LIN {X 0,Y 740.336,Z 905.286,A -85,B 0,C 180,E1 33713.646,E2 33713.646} C_VEL
LIN {X 0,Y 741.074,Z 665.697,A -85,B 0,C 180,E1 33710.789,E2 33710.789} C_VEL
LIN {X 0,Y 741.733,Z 456.435,A -85,B 0,C 180,E1 33708.221,E2 33708.221} C_VEL
LIN {X 0,Y 741.657,Z 433.468,A -85,B 0,C 180,E1 33707.923,E2 33707.923} C_VEL
LIN {X 0,Y 740.112,Z 427.36,A -85,B 0,C 180,E1 33707.725,E2 33707.725} C_VEL
LIN {X 0,Y 740.318,Z 399.493,A -85,B 0,C 180,E1 33705.878,E2 33705.878} C_VEL
LIN {X 0,Y 737.201,Z 392.802,A -85,B 0,C 180,E1 33705.183,E2 33705.183} C_VEL
LIN {X 0,Y 736.058,Z 389.544,A -85,B 0,C 180,E1 33704.846,E2 33704.846} C_VEL
LIN {X 0,Y 736.094,Z 389.54,A -85,B 0,C 180,E1 33701.833,E2 33701.833} C_VEL
LIN {X 0,Y 736.034,Z 389.542,A -85,B 0,C 180,E1 33699.075,E2 33699.075} C_VEL
LIN {X 0,Y 736.07,Z 389.535,A -85,B 0,C 180,E1 33696.415,E2 33696.415} C_VEL
LIN {X 0,Y 736.045,Z 389.543,A -85,B 0,C 180,E1 33693.349,E2 33693.349} C_VEL
LIN {X 0,Y 736.022,Z 389.539,A -85,B 0,C 180,E1 33690.808,E2 33690.808} C_VEL
LIN {X 0,Y 736.056,Z 389.537,A -85,B 0,C 180,E1 33688.212,E2 33688.212} C_VEL
LIN {X 0,Y 736.036,Z 389.54,A -85,B 0,C 180,E1 33685.164,E2 33685.164} C_VEL
LIN {X 0,Y 736.009,Z 389.543,A -85,B 0,C 180,E1 33682.695,E2 33682.695} C_VEL
LIN {X 0,Y 736.01,Z 389.536,A -85,B 0,C 180,E1 33680.352,E2 33680.352} C_VEL
LIN {X 0,Y 736.099,Z 389.541,A -85,B 0,C 180,E1 33677.55,E2 33677.55} C_VEL
LIN {X 0,Y 736.004,Z 389.539,A -85,B 0,C 180,E1 33674.717,E2 33674.717} C_VEL
LIN {X 0,Y 735.992,Z 389.544,A -85,B 0,C 180,E1 33672.475,E2 33672.475} C_VEL
LIN {X 0,Y 735.989,Z 389.542,A -85,B 0,C 180,E1 33670.173,E2 33670.173} C_VEL
LIN {X 0,Y 736.026,Z 389.541,A -85,B 0,C 180,E1 33667.651,E2 33667.651} C_VEL
LIN {X 0,Y 736.016,Z 389.541,A -85,B 0,C 180,E1 33664.675,E2 33664.675} C_VEL
LIN {X 0,Y 735.992,Z 389.54,A -85,B 0,C 180,E1 33662.258,E2 33662.258} C_VEL
LIN {X 0,Y 735.996,Z 389.544,A -85,B 0,C 180,E1 33660,E2 33660} C_VEL
LIN {X 0,Y 736.012,Z 389.54,A -85,B 0,C 180,E1 33657.664,E2 33657.664} C_VEL
LIN {X 0,Y 736.088,Z 389.541,A -85,B 0,C 180,E1 33654.778,E2 33654.778} C_VEL
LIN {X 0,Y 736.012,Z 389.538,A -85,B 0,C 180,E1 33652.035,E2 33652.035} C_VEL
LIN {X 0,Y 736.014,Z 389.539,A -85,B 0,C 180,E1 33649.67,E2 33649.67} C_VEL
LIN {X 0,Y 736.089,Z 389.542,A -85,B 0,C 180,E1 33648.953,E2 33648.953} C_VEL
LIN {X 0,Y 735.153,Z 389.668,A -85,B 0,C 180,E1 33648.354,E2 33648.354} C_VEL
LIN {X 0,Y 728.691,Z 390.459,A -85,B 0,C 180,E1 33646.675,E2 33646.675} C_VEL
LIN {X 0,Y 728.114,Z 390.522,A -85,B 0,C 180,E1 33646.239,E2 33646.239} C_VEL
LIN {X 0,Y 728.083,Z 390.527,A -85,B 0,C 180,E1 33643.648,E2 33643.648} C_VEL
LIN {X 0,Y 728.114,Z 390.532,A -85,B 0,C 180,E1 33641.089,E2 33641.089} C_VEL
LIN {X 0,Y 728.117,Z 390.526,A -85,B 0,C 180,E1 33637.946,E2 33637.946} C_VEL
LIN {X 0,Y 728.097,Z 390.528,A -85,B 0,C 180,E1 33635.324,E2 33635.324} C_VEL
LIN {X 0,Y 728.159,Z 390.532,A -85,B 0,C 180,E1 33632.493,E2 33632.493} C_VEL
LIN {X 0,Y 728.112,Z 390.518,A -85,B 0,C 180,E1 33629.553,E2 33629.553} C_VEL
LIN {X 0,Y 728.12,Z 390.532,A -85,B 0,C 180,E1 33626.869,E2 33626.869} C_VEL
LIN {X 0,Y 728.157,Z 390.525,A -85,B 0,C 180,E1 33623.907,E2 33623.907} C_VEL
LIN {X 0,Y 728.115,Z 390.52,A -85,B 0,C 180,E1 33621.126,E2 33621.126} C_VEL
LIN {X 0,Y 728.16,Z 390.533,A -85,B 0,C 180,E1 33618.322,E2 33618.322} C_VEL
LIN {X 0,Y 728.142,Z 390.527,A -85,B 0,C 180,E1 33615.325,E2 33615.325} C_VEL
LIN {X 0,Y 728.178,Z 390.706,A -85,B 0,C 180,E1 33613.598,E2 33613.598} C_VEL
LIN {X 0,Y 731.353,Z 398.193,A -85,B 0,C 180,E1 33612.834,E2 33612.834} C_VEL
LIN {X 0,Y 735.188,Z 404.542,A -85,B 0,C 180,E1 33612.475,E2 33612.475} C_VEL
LIN {X 0,Y 735.82,Z 407.925,A -85,B 0,C 180,E1 33612.386,E2 33612.386} C_VEL
LIN {X 0,Y 734.951,Z 615.725,A -85,B 0,C 180,E1 33609.805,E2 33609.805} C_VEL
LIN {X 0,Y 734.065,Z 840.668,A -85,B 0,C 180,E1 33607.107,E2 33607.107} C_VEL
LIN {X 0,Y 733.846,Z 880.574,A -85,B 0,C 180,E1 33606.601,E2 33606.601} C_VEL
LIN {X 0,Y 733.519,Z 907.444,A -85,B 0,C 180,E1 33606.104,E2 33606.104} C_VEL
LIN {X 0,Y 733.177,Z 933.426,A -85,B 0,C 180,E1 33605.468,E2 33605.468} C_VEL
LIN {X 0,Y 732.752,Z 961.422,A -85,B 0,C 180,E1 33604.607,E2 33604.607} C_VEL
LIN {X 0,Y 732.215,Z 986.668,A -85,B 0,C 180,E1 33603.664,E2 33603.664} C_VEL
LIN {X 0,Y 731.798,Z 1007.845,A -85,B 0,C 180,E1 33602.75,E2 33602.75} C_VEL
LIN {X 0,Y 731.38,Z 1029.215,A -85,B 0,C 180,E1 33601.706,E2 33601.706} C_VEL
LIN {X 0,Y 730.847,Z 1054.293,A -85,B 0,C 180,E1 33600.312,E2 33600.312} C_VEL
LIN {X 0,Y 730.374,Z 1074.643,A -85,B 0,C 180,E1 33599.027,E2 33599.027} C_VEL
LIN {X 0,Y 730.005,Z 1092.923,A -85,B 0,C 180,E1 33597.75,E2 33597.75} C_VEL
LIN {X 0,Y 729.604,Z 1114.26,A -85,B 0,C 180,E1 33596.093,E2 33596.093} C_VEL
LIN {X 0,Y 729.199,Z 1132.017,A -85,B 0,C 180,E1 33594.544,E2 33594.544} C_VEL
LIN {X 0,Y 728.96,Z 1147.136,A -85,B 0,C 180,E1 33593.092,E2 33593.092} C_VEL
LIN {X 0,Y 728.695,Z 1164.65,A -85,B 0,C 180,E1 33591.233,E2 33591.233} C_VEL
LIN {X 0,Y 728.444,Z 1179.846,A -85,B 0,C 180,E1 33589.396,E2 33589.396} C_VEL
LIN {X 0,Y 728.269,Z 1191.551,A -85,B 0,C 180,E1 33587.824,E2 33587.824} C_VEL
LIN {X 0,Y 728.153,Z 1202.004,A -85,B 0,C 180,E1 33586.263,E2 33586.263} C_VEL
LIN {X 0,Y 728.097,Z 1212.225,A -85,B 0,C 180,E1 33584.551,E2 33584.551} C_VEL
LIN {X 0,Y 728.002,Z 1223.462,A -85,B 0,C 180,E1 33582.368,E2 33582.368} C_VEL
LIN {X 0,Y 727.957,Z 1231.704,A -85,B 0,C 180,E1 33580.431,E2 33580.431} C_VEL
LIN {X 0,Y 727.92,Z 1237.917,A -85,B 0,C 180,E1 33578.686,E2 33578.686} C_VEL
LIN {X 0,Y 727.914,Z 1243.464,A -85,B 0,C 180,E1 33576.78,E2 33576.78} C_VEL
LIN {X 0,Y 727.907,Z 1247.988,A -85,B 0,C 180,E1 33574.645,E2 33574.645} C_VEL
LIN {X 0,Y 727.907,Z 1250.641,A -85,B 0,C 180,E1 33572.594,E2 33572.594} C_VEL
LIN {X 0,Y 727.869,Z 1251.748,A -85,B 0,C 180,E1 33570.862,E2 33570.862} C_VEL
LIN {X 0,Y 727.863,Z 1251.816,A -85,B 0,C 180,E1 33569.288,E2 33569.288} C_VEL
LIN {X 0,Y 727.903,Z 1250.914,A -85,B 0,C 180,E1 33567.635,E2 33567.635} C_VEL
LIN {X 0,Y 727.919,Z 1248.744,A -85,B 0,C 180,E1 33565.743,E2 33565.743} C_VEL
LIN {X 0,Y 727.926,Z 1244.646,A -85,B 0,C 180,E1 33563.609,E2 33563.609} C_VEL
LIN {X 0,Y 727.938,Z 1238.951,A -85,B 0,C 180,E1 33561.545,E2 33561.545} C_VEL
LIN {X 0,Y 727.959,Z 1232.899,A -85,B 0,C 180,E1 33559.791,E2 33559.791} C_VEL
LIN {X 0,Y 727.968,Z 1225.974,A -85,B 0,C 180,E1 33558.107,E2 33558.107} C_VEL
LIN {X 0,Y 727.992,Z 1218.275,A -85,B 0,C 180,E1 33556.494,E2 33556.494} C_VEL
LIN {X 0,Y 728.087,Z 1209.438,A -85,B 0,C 180,E1 33554.872,E2 33554.872} C_VEL
LIN {X 0,Y 728.235,Z 1197.825,A -85,B 0,C 180,E1 33552.992,E2 33552.992} C_VEL
LIN {X 0,Y 728.407,Z 1183.707,A -85,B 0,C 180,E1 33551.012,E2 33551.012} C_VEL
LIN {X 0,Y 728.579,Z 1170.319,A -85,B 0,C 180,E1 33549.345,E2 33549.345} C_VEL
LIN {X 0,Y 728.783,Z 1156.105,A -85,B 0,C 180,E1 33547.746,E2 33547.746} C_VEL
LIN {X 0,Y 729.15,Z 1137.559,A -85,B 0,C 180,E1 33545.878,E2 33545.878} C_VEL
LIN {X 0,Y 729.432,Z 1120.293,A -85,B 0,C 180,E1 33544.329,E2 33544.329} C_VEL
LIN {X 0,Y 729.793,Z 1103.261,A -85,B 0,C 180,E1 33542.941,E2 33542.941} C_VEL
LIN {X 0,Y 730.277,Z 1081.154,A -85,B 0,C 180,E1 33541.319,E2 33541.319} C_VEL
LIN {X 0,Y 730.68,Z 1060.659,A -85,B 0,C 180,E1 33539.987,E2 33539.987} C_VEL
LIN {X 0,Y 731.098,Z 1040.76,A -85,B 0,C 180,E1 33538.823,E2 33538.823} C_VEL
LIN {X 0,Y 731.664,Z 1017.402,A -85,B 0,C 180,E1 33537.606,E2 33537.606} C_VEL
LIN {X 0,Y 732.144,Z 991.959,A -85,B 0,C 180,E1 33536.464,E2 33536.464} C_VEL
LIN {X 0,Y 732.524,Z 970.715,A -85,B 0,C 180,E1 33535.636,E2 33535.636} C_VEL
LIN {X 0,Y 732.881,Z 949.473,A -85,B 0,C 180,E1 33534.918,E2 33534.918} C_VEL
LIN {X 0,Y 733.282,Z 925.666,A -85,B 0,C 180,E1 33534.236,E2 33534.236} C_VEL
LIN {X 0,Y 733.637,Z 898.906,A -85,B 0,C 180,E1 33533.631,E2 33533.631} C_VEL
LIN {X 0,Y 733.897,Z 872.286,A -85,B 0,C 180,E1 33533.187,E2 33533.187} C_VEL
LIN {X 0,Y 734.857,Z 637.491,A -85,B 0,C 180,E1 33530.37,E2 33530.37} C_VEL
LIN {X 0,Y 735.731,Z 430.486,A -85,B 0,C 180,E1 33527.809,E2 33527.809} C_VEL
LIN {X 0,Y 735.653,Z 406.249,A -85,B 0,C 180,E1 33527.491,E2 33527.491} C_VEL
LIN {X 0,Y 734.384,Z 402.855,A -85,B 0,C 180,E1 33527.356,E2 33527.356} C_VEL
LIN {X 0,Y 731.047,Z 397.734,A -85,B 0,C 180,E1 33527.033,E2 33527.033} C_VEL
LIN {X 0,Y 728.173,Z 390.725,A -85,B 0,C 180,E1 33526.313,E2 33526.313} C_VEL
LIN {X 0,Y 728.153,Z 390.533,A -85,B 0,C 180,E1 33523.361,E2 33523.361} C_VEL
LIN {X 0,Y 728.159,Z 390.522,A -85,B 0,C 180,E1 33520.298,E2 33520.298} C_VEL
LIN {X 0,Y 728.155,Z 390.532,A -85,B 0,C 180,E1 33517.207,E2 33517.207} C_VEL
LIN {X 0,Y 728.16,Z 390.515,A -85,B 0,C 180,E1 33514.102,E2 33514.102} C_VEL
LIN {X 0,Y 728.159,Z 390.525,A -85,B 0,C 180,E1 33510.994,E2 33510.994} C_VEL
LIN {X 0,Y 728.159,Z 390.52,A -85,B 0,C 180,E1 33507.921,E2 33507.921} C_VEL
LIN {X 0,Y 728.153,Z 390.524,A -85,B 0,C 180,E1 33504.813,E2 33504.813} C_VEL
LIN {X 0,Y 728.154,Z 390.518,A -85,B 0,C 180,E1 33501.678,E2 33501.678} C_VEL
LIN {X 0,Y 728.15,Z 390.527,A -85,B 0,C 180,E1 33498.646,E2 33498.646} C_VEL
LIN {X 0,Y 728.156,Z 390.515,A -85,B 0,C 180,E1 33495.613,E2 33495.613} C_VEL
LIN {X 0,Y 728.131,Z 390.526,A -85,B 0,C 180,E1 33492.692,E2 33492.692} C_VEL
LIN {X 0,Y 728.142,Z 390.519,A -85,B 0,C 180,E1 33489.804,E2 33489.804} C_VEL
LIN {X 0,Y 728.134,Z 390.521,A -85,B 0,C 180,E1 33486.941,E2 33486.941} C_VEL
LIN {X 0,Y 728.153,Z 390.527,A -85,B 0,C 180,E1 33484.016,E2 33484.016} C_VEL
LIN {X 0,Y 728.153,Z 390.519,A -85,B 0,C 180,E1 33480.944,E2 33480.944} C_VEL
LIN {X 0,Y 728.14,Z 390.531,A -85,B 0,C 180,E1 33477.954,E2 33477.954} C_VEL
LIN {X 0,Y 728.157,Z 390.519,A -85,B 0,C 180,E1 33474.879,E2 33474.879} C_VEL
LIN {X 0,Y 728.121,Z 390.526,A -85,B 0,C 180,E1 33472.027,E2 33472.027} C_VEL
LIN {X 0,Y 728.149,Z 390.528,A -85,B 0,C 180,E1 33469.156,E2 33469.156} C_VEL
LIN {X 0,Y 728.132,Z 390.52,A -85,B 0,C 180,E1 33466.257,E2 33466.257} C_VEL
LIN {X 0,Y 728.138,Z 390.527,A -85,B 0,C 180,E1 33463.403,E2 33463.403} C_VEL
LIN {X 0,Y 728.157,Z 390.514,A -85,B 0,C 180,E1 33460.34,E2 33460.34} C_VEL
LIN {X 0,Y 728.119,Z 390.528,A -85,B 0,C 180,E1 33457.472,E2 33457.472} C_VEL
LIN {X 0,Y 728.152,Z 390.524,A -85,B 0,C 180,E1 33454.631,E2 33454.631} C_VEL
LIN {X 0,Y 728.125,Z 390.524,A -85,B 0,C 180,E1 33451.721,E2 33451.721} C_VEL
LIN {X 0,Y 728.13,Z 390.527,A -85,B 0,C 180,E1 33448.913,E2 33448.913} C_VEL
LIN {X 0,Y 728.158,Z 390.519,A -85,B 0,C 180,E1 33445.831,E2 33445.831} C_VEL
LIN {X 0,Y 728.11,Z 390.528,A -85,B 0,C 180,E1 33443.023,E2 33443.023} C_VEL
LIN {X 0,Y 728.158,Z 390.53,A -85,B 0,C 180,E1 33440.215,E2 33440.215} C_VEL
LIN {X 0,Y 728.127,Z 390.529,A -85,B 0,C 180,E1 33437.282,E2 33437.282} C_VEL
LIN {X 0,Y 728.174,Z 390.66,A -85,B 0,C 180,E1 33435.678,E2 33435.678} C_VEL
LIN {X 0,Y 729.538,Z 394.152,A -85,B 0,C 180,E1 33435.323,E2 33435.323} C_VEL
LIN {X 0,Y 733.944,Z 403.814,A -85,B 0,C 180,E1 33434.309,E2 33434.309} C_VEL
LIN {X 0,Y 733.709,Z 428.121,A -85,B 0,C 180,E1 33432.709,E2 33432.709} C_VEL
LIN {X 0,Y 735.845,Z 436.973,A -85,B 0,C 180,E1 33432.441,E2 33432.441} C_VEL
LIN {X 0,Y 734.928,Z 651.151,A -85,B 0,C 180,E1 33429.784,E2 33429.784} C_VEL
LIN {X 0,Y 734.041,Z 876.977,A -85,B 0,C 180,E1 33427.077,E2 33427.077} C_VEL
LIN {X 0,Y 733.835,Z 912.252,A -85,B 0,C 180,E1 33426.621,E2 33426.621} C_VEL
LIN {X 0,Y 733.505,Z 939.344,A -85,B 0,C 180,E1 33426.107,E2 33426.107} C_VEL
LIN {X 0,Y 733.142,Z 965.257,A -85,B 0,C 180,E1 33425.463,E2 33425.463} C_VEL
LIN {X 0,Y 732.696,Z 993.123,A -85,B 0,C 180,E1 33424.592,E2 33424.592} C_VEL
LIN {X 0,Y 732.21,Z 1016.791,A -85,B 0,C 180,E1 33423.704,E2 33423.704} C_VEL
LIN {X 0,Y 731.802,Z 1037.53,A -85,B 0,C 180,E1 33422.81,E2 33422.81} C_VEL
LIN {X 0,Y 731.394,Z 1058.143,A -85,B 0,C 180,E1 33421.806,E2 33421.806} C_VEL
LIN {X 0,Y 730.878,Z 1083.375,A -85,B 0,C 180,E1 33420.412,E2 33420.412} C_VEL
LIN {X 0,Y 730.405,Z 1103.558,A -85,B 0,C 180,E1 33419.144,E2 33419.144} C_VEL
LIN {X 0,Y 730.02,Z 1121.613,A -85,B 0,C 180,E1 33417.89,E2 33417.89} C_VEL
LIN {X 0,Y 729.65,Z 1141.908,A -85,B 0,C 180,E1 33416.334,E2 33416.334} C_VEL
LIN {X 0,Y 729.214,Z 1161.485,A -85,B 0,C 180,E1 33414.638,E2 33414.638} C_VEL
LIN {X 0,Y 728.956,Z 1177.508,A -85,B 0,C 180,E1 33413.1,E2 33413.1} C_VEL
LIN {X 0,Y 728.685,Z 1194.964,A -85,B 0,C 180,E1 33411.241,E2 33411.241} C_VEL
LIN {X 0,Y 728.438,Z 1210.135,A -85,B 0,C 180,E1 33409.404,E2 33409.404} C_VEL
LIN {X 0,Y 728.265,Z 1221.814,A -85,B 0,C 180,E1 33407.831,E2 33407.831} C_VEL
LIN {X 0,Y 728.149,Z 1232.764,A -85,B 0,C 180,E1 33406.189,E2 33406.189} C_VEL
LIN {X 0,Y 728.085,Z 1244.291,A -85,B 0,C 180,E1 33404.233,E2 33404.233} C_VEL
LIN {X 0,Y 727.974,Z 1254.701,A -85,B 0,C 180,E1 33402.134,E2 33402.134} C_VEL
LIN {X 0,Y 727.957,Z 1261.876,A -85,B 0,C 180,E1 33400.431,E2 33400.431} C_VEL
LIN {X 0,Y 727.915,Z 1267.782,A -85,B 0,C 180,E1 33398.773,E2 33398.773} C_VEL
LIN {X 0,Y 727.919,Z 1273.167,A -85,B 0,C 180,E1 33396.946,E2 33396.946} C_VEL
LIN {X 0,Y 727.911,Z 1277.776,A -85,B 0,C 180,E1 33394.81,E2 33394.81} C_VEL
LIN {X 0,Y 727.914,Z 1280.538,A -85,B 0,C 180,E1 33392.759,E2 33392.759} C_VEL
LIN {X 0,Y 727.874,Z 1281.714,A -85,B 0,C 180,E1 33391.027,E2 33391.027} C_VEL
LIN {X 0,Y 727.863,Z 1281.828,A -85,B 0,C 180,E1 33389.374,E2 33389.374} C_VEL
LIN {X 0,Y 727.907,Z 1280.949,A -85,B 0,C 180,E1 33387.721,E2 33387.721} C_VEL
LIN {X 0,Y 727.919,Z 1278.809,A -85,B 0,C 180,E1 33385.829,E2 33385.829} C_VEL
LIN {X 0,Y 727.926,Z 1274.743,A -85,B 0,C 180,E1 33383.695,E2 33383.695} C_VEL
LIN {X 0,Y 727.939,Z 1269.086,A -85,B 0,C 180,E1 33381.632,E2 33381.632} C_VEL
LIN {X 0,Y 727.958,Z 1263.061,A -85,B 0,C 180,E1 33379.878,E2 33379.878} C_VEL
LIN {X 0,Y 727.966,Z 1256.163,A -85,B 0,C 180,E1 33378.195,E2 33378.195} C_VEL
LIN {X 0,Y 727.992,Z 1248.905,A -85,B 0,C 180,E1 33376.663,E2 33376.663} C_VEL
LIN {X 0,Y 728.086,Z 1240.621,A -85,B 0,C 180,E1 33375.124,E2 33375.124} C_VEL
LIN {X 0,Y 728.176,Z 1230.723,A -85,B 0,C 180,E1 33373.491,E2 33373.491} C_VEL
LIN {X 0,Y 728.346,Z 1218.375,A -85,B 0,C 180,E1 33371.682,E2 33371.682} C_VEL
LIN {X 0,Y 728.544,Z 1202.255,A -85,B 0,C 180,E1 33369.617,E2 33369.617} C_VEL
LIN {X 0,Y 728.751,Z 1188.102,A -85,B 0,C 180,E1 33368.007,E2 33368.007} C_VEL
LIN {X 0,Y 729.047,Z 1172.215,A -85,B 0,C 180,E1 33366.372,E2 33366.372} C_VEL
LIN {X 0,Y 729.421,Z 1152.323,A -85,B 0,C 180,E1 33364.548,E2 33364.548} C_VEL
LIN {X 0,Y 729.732,Z 1135.012,A -85,B 0,C 180,E1 33363.123,E2 33363.123} C_VEL
LIN {X 0,Y 730.171,Z 1116.028,A -85,B 0,C 180,E1 33361.706,E2 33361.706} C_VEL
LIN {X 0,Y 730.667,Z 1092.249,A -85,B 0,C 180,E1 33360.13,E2 33360.13} C_VEL
LIN {X 0,Y 731.055,Z 1072.524,A -85,B 0,C 180,E1 33358.966,E2 33358.966} C_VEL
LIN {X 0,Y 731.511,Z 1052.074,A -85,B 0,C 180,E1 33357.885,E2 33357.885} C_VEL
LIN {X 0,Y 732.097,Z 1026.682,A -85,B 0,C 180,E1 33356.705,E2 33356.705} C_VEL
LIN {X 0,Y 732.513,Z 1002.281,A -85,B 0,C 180,E1 33355.738,E2 33355.738} C_VEL
LIN {X 0,Y 732.868,Z 981.29,A -85,B 0,C 180,E1 33355.021,E2 33355.021} C_VEL
LIN {X 0,Y 733.241,Z 958.436,A -85,B 0,C 180,E1 33354.353,E2 33354.353} C_VEL
LIN {X 0,Y 733.618,Z 931.508,A -85,B 0,C 180,E1 33353.727,E2 33353.727} C_VEL
LIN {X 0,Y 733.884,Z 903.946,A -85,B 0,C 180,E1 33353.255,E2 33353.255} C_VEL
LIN {X 0,Y 734.857,Z 667.784,A -85,B 0,C 180,E1 33350.418,E2 33350.418} C_VEL
LIN {X 0,Y 735.744,Z 458.714,A -85,B 0,C 180,E1 33347.833,E2 33347.833} C_VEL
LIN {X 0,Y 735.67,Z 435.525,A -85,B 0,C 180,E1 33347.527,E2 33347.527} C_VEL
LIN {X 0,Y 733.585,Z 427.36,A -85,B 0,C 180,E1 33347.259,E2 33347.259} C_VEL
LIN {X 0,Y 733.862,Z 403.52,A -85,B 0,C 180,E1 33345.664,E2 33345.664} C_VEL
LIN {X 0,Y 728.311,Z 391.368,A -85,B 0,C 180,E1 33344.383,E2 33344.383} C_VEL
LIN {X 0,Y 728.158,Z 390.532,A -85,B 0,C 180,E1 33344.282,E2 33344.282} C_VEL
LIN {X 0,Y 728.11,Z 390.525,A -85,B 0,C 180,E1 33341.436,E2 33341.436} C_VEL
LIN {X 0,Y 728.104,Z 390.529,A -85,B 0,C 180,E1 33338.772,E2 33338.772} C_VEL
LIN {X 0,Y 728.16,Z 390.529,A -85,B 0,C 180,E1 33335.898,E2 33335.898} C_VEL
LIN {X 0,Y 728.09,Z 390.53,A -85,B 0,C 180,E1 33333.112,E2 33333.112} C_VEL
LIN {X 0,Y 728.092,Z 390.527,A -85,B 0,C 180,E1 33330.577,E2 33330.577} C_VEL
LIN {X 0,Y 728.161,Z 390.531,A -85,B 0,C 180,E1 33327.677,E2 33327.677} C_VEL
LIN {X 0,Y 728.079,Z 390.527,A -85,B 0,C 180,E1 33324.936,E2 33324.936} C_VEL
LIN {X 0,Y 728.071,Z 390.531,A -85,B 0,C 180,E1 33322.53,E2 33322.53} C_VEL
LIN {X 0,Y 728.117,Z 390.522,A -85,B 0,C 180,E1 33319.912,E2 33319.912} C_VEL
LIN {X 0,Y 728.083,Z 390.532,A -85,B 0,C 180,E1 33316.927,E2 33316.927} C_VEL
LIN {X 0,Y 728.058,Z 390.526,A -85,B 0,C 180,E1 33314.51,E2 33314.51} C_VEL
LIN {X 0,Y 728.056,Z 390.533,A -85,B 0,C 180,E1 33312.21,E2 33312.21} C_VEL
LIN {X 0,Y 728.112,Z 390.53,A -85,B 0,C 180,E1 33309.565,E2 33309.565} C_VEL
LIN {X 0,Y 728.064,Z 390.534,A -85,B 0,C 180,E1 33306.625,E2 33306.625} C_VEL
LIN {X 0,Y 728.05,Z 390.529,A -85,B 0,C 180,E1 33304.253,E2 33304.253} C_VEL
LIN {X 0,Y 728.054,Z 390.529,A -85,B 0,C 180,E1 33301.968,E2 33301.968} C_VEL
LIN {X 0,Y 728.098,Z 390.534,A -85,B 0,C 180,E1 33299.449,E2 33299.449} C_VEL
LIN {X 0,Y 728.091,Z 390.526,A -85,B 0,C 180,E1 33296.457,E2 33296.457} C_VEL
LIN {X 0,Y 728.068,Z 390.532,A -85,B 0,C 180,E1 33294.009,E2 33294.009} C_VEL
LIN {X 0,Y 728.075,Z 390.527,A -85,B 0,C 180,E1 33291.629,E2 33291.629} C_VEL
LIN {X 0,Y 728.161,Z 390.532,A -85,B 0,C 180,E1 33288.836,E2 33288.836} C_VEL
LIN {X 0,Y 728.114,Z 390.522,A -85,B 0,C 180,E1 33286.239,E2 33286.239} C_VEL
LIN {X 0,Y 727.075,Z 390.651,A -85,B 0,C 180,E1 33285.633,E2 33285.633} C_VEL
LIN {X 0,Y 720.662,Z 391.451,A -85,B 0,C 180,E1 33283.934,E2 33283.934} C_VEL
LIN {X 0,Y 720.147,Z 391.516,A -85,B 0,C 180,E1 33283.493,E2 33283.493} C_VEL
LIN {X 0,Y 720.219,Z 391.512,A -85,B 0,C 180,E1 33280.706,E2 33280.706} C_VEL
LIN {X 0,Y 720.166,Z 391.516,A -85,B 0,C 180,E1 33277.812,E2 33277.812} C_VEL
LIN {X 0,Y 720.161,Z 391.517,A -85,B 0,C 180,E1 33275.209,E2 33275.209} C_VEL
LIN {X 0,Y 720.218,Z 391.518,A -85,B 0,C 180,E1 33272.329,E2 33272.329} C_VEL
LIN {X 0,Y 720.169,Z 391.506,A -85,B 0,C 180,E1 33269.459,E2 33269.459} C_VEL
LIN {X 0,Y 720.199,Z 391.523,A -85,B 0,C 180,E1 33266.686,E2 33266.686} C_VEL
LIN {X 0,Y 720.195,Z 391.515,A -85,B 0,C 180,E1 33263.543,E2 33263.543} C_VEL
LIN {X 0,Y 720.194,Z 391.513,A -85,B 0,C 180,E1 33260.643,E2 33260.643} C_VEL
LIN {X 0,Y 720.215,Z 391.513,A -85,B 0,C 180,E1 33257.567,E2 33257.567} C_VEL
LIN {X 0,Y 720.188,Z 391.524,A -85,B 0,C 180,E1 33254.696,E2 33254.696} C_VEL
LIN {X 0,Y 720.236,Z 391.672,A -85,B 0,C 180,E1 33254.131,E2 33254.131} C_VEL
LIN {X 0,Y 721.542,Z 395.043,A -85,B 0,C 180,E1 33253.781,E2 33253.781} C_VEL
LIN {X 0,Y 723.12,Z 398.553,A -85,B 0,C 180,E1 33253.438,E2 33253.438} C_VEL
LIN {X 0,Y 729.888,Z 409.055,A -85,B 0,C 180,E1 33252.798,E2 33252.798} C_VEL
LIN {X 0,Y 728.802,Z 615.141,A -85,B 0,C 180,E1 33250.217,E2 33250.217} C_VEL
LIN {X 0,Y 727.684,Z 839.955,A -85,B 0,C 180,E1 33247.497,E2 33247.497} C_VEL
LIN {X 0,Y 727.403,Z 880.724,A -85,B 0,C 180,E1 33246.978,E2 33246.978} C_VEL
LIN {X 0,Y 726.998,Z 907.88,A -85,B 0,C 180,E1 33246.47,E2 33246.47} C_VEL
LIN {X 0,Y 726.57,Z 933.577,A -85,B 0,C 180,E1 33245.836,E2 33245.836} C_VEL
LIN {X 0,Y 726.058,Z 960.87,A -85,B 0,C 180,E1 33244.994,E2 33244.994} C_VEL
LIN {X 0,Y 725.384,Z 986.687,A -85,B 0,C 180,E1 33244.024,E2 33244.024} C_VEL
LIN {X 0,Y 724.841,Z 1007.861,A -85,B 0,C 180,E1 33243.105,E2 33243.105} C_VEL
LIN {X 0,Y 724.295,Z 1030.12,A -85,B 0,C 180,E1 33242.007,E2 33242.007} C_VEL
LIN {X 0,Y 723.601,Z 1055.717,A -85,B 0,C 180,E1 33240.559,E2 33240.559} C_VEL
LIN {X 0,Y 723.046,Z 1075.315,A -85,B 0,C 180,E1 33239.304,E2 33239.304} C_VEL
LIN {X 0,Y 722.545,Z 1094.746,A -85,B 0,C 180,E1 33237.927,E2 33237.927} C_VEL
LIN {X 0,Y 721.991,Z 1116.685,A -85,B 0,C 180,E1 33236.178,E2 33236.178} C_VEL
LIN {X 0,Y 721.541,Z 1133.318,A -85,B 0,C 180,E1 33234.7,E2 33234.7} C_VEL
LIN {X 0,Y 721.216,Z 1149.701,A -85,B 0,C 180,E1 33233.095,E2 33233.095} C_VEL
LIN {X 0,Y 720.843,Z 1167.498,A -85,B 0,C 180,E1 33231.135,E2 33231.135} C_VEL
LIN {X 0,Y 720.574,Z 1181.141,A -85,B 0,C 180,E1 33229.448,E2 33229.448} C_VEL
LIN {X 0,Y 720.364,Z 1192.721,A -85,B 0,C 180,E1 33227.859,E2 33227.859} C_VEL
LIN {X 0,Y 720.21,Z 1204.621,A -85,B 0,C 180,E1 33226.033,E2 33226.033} C_VEL
LIN {X 0,Y 720.069,Z 1216.629,A -85,B 0,C 180,E1 33223.895,E2 33223.895} C_VEL
LIN {X 0,Y 719.991,Z 1225.252,A -85,B 0,C 180,E1 33222.1,E2 33222.1} C_VEL
LIN {X 0,Y 719.97,Z 1232.279,A -85,B 0,C 180,E1 33220.397,E2 33220.397} C_VEL
LIN {X 0,Y 719.924,Z 1238.175,A -85,B 0,C 180,E1 33218.703,E2 33218.703} C_VEL
LIN {X 0,Y 719.917,Z 1243.661,A -85,B 0,C 180,E1 33216.776,E2 33216.776} C_VEL
LIN {X 0,Y 719.908,Z 1247.989,A -85,B 0,C 180,E1 33214.696,E2 33214.696} C_VEL
LIN {X 0,Y 719.908,Z 1250.641,A -85,B 0,C 180,E1 33212.623,E2 33212.623} C_VEL
LIN {X 0,Y 719.87,Z 1251.748,A -85,B 0,C 180,E1 33210.872,E2 33210.872} C_VEL
LIN {X 0,Y 719.863,Z 1251.816,A -85,B 0,C 180,E1 33209.28,E2 33209.28} C_VEL
LIN {X 0,Y 719.903,Z 1250.914,A -85,B 0,C 180,E1 33207.608,E2 33207.608} C_VEL
LIN {X 0,Y 719.918,Z 1248.743,A -85,B 0,C 180,E1 33205.695,E2 33205.695} C_VEL
LIN {X 0,Y 719.926,Z 1244.645,A -85,B 0,C 180,E1 33203.537,E2 33203.537} C_VEL
LIN {X 0,Y 719.944,Z 1238.919,A -85,B 0,C 180,E1 33201.441,E2 33201.441} C_VEL
LIN {X 0,Y 719.97,Z 1232.898,A -85,B 0,C 180,E1 33199.676,E2 33199.676} C_VEL
LIN {X 0,Y 719.988,Z 1226.33,A -85,B 0,C 180,E1 33198.055,E2 33198.055} C_VEL
LIN {X 0,Y 720.024,Z 1219.095,A -85,B 0,C 180,E1 33196.506,E2 33196.506} C_VEL
LIN {X 0,Y 720.131,Z 1210.833,A -85,B 0,C 180,E1 33194.948,E2 33194.948} C_VEL
LIN {X 0,Y 720.27,Z 1200.959,A -85,B 0,C 180,E1 33193.297,E2 33193.297} C_VEL
LIN {X 0,Y 720.466,Z 1188.635,A -85,B 0,C 180,E1 33191.466,E2 33191.466} C_VEL
LIN {X 0,Y 720.732,Z 1172.449,A -85,B 0,C 180,E1 33189.364,E2 33189.364} C_VEL
LIN {X 0,Y 720.986,Z 1158.442,A -85,B 0,C 180,E1 33187.75,E2 33187.75} C_VEL
LIN {X 0,Y 721.332,Z 1143.49,A -85,B 0,C 180,E1 33186.188,E2 33186.188} C_VEL
LIN {X 0,Y 721.81,Z 1123.333,A -85,B 0,C 180,E1 33184.302,E2 33184.302} C_VEL
LIN {X 0,Y 722.249,Z 1105.47,A -85,B 0,C 180,E1 33182.813,E2 33182.813} C_VEL
LIN {X 0,Y 722.764,Z 1086.774,A -85,B 0,C 180,E1 33181.399,E2 33181.399} C_VEL
LIN {X 0,Y 723.393,Z 1062.835,A -85,B 0,C 180,E1 33179.791,E2 33179.791} C_VEL
LIN {X 0,Y 723.928,Z 1042.439,A -85,B 0,C 180,E1 33178.576,E2 33178.576} C_VEL
LIN {X 0,Y 724.507,Z 1021.941,A -85,B 0,C 180,E1 33177.484,E2 33177.484} C_VEL
LIN {X 0,Y 725.211,Z 996.422,A -85,B 0,C 180,E1 33176.291,E2 33176.291} C_VEL
LIN {X 0,Y 725.73,Z 971.973,A -85,B 0,C 180,E1 33175.316,E2 33175.316} C_VEL
LIN {X 0,Y 726.176,Z 951.16,A -85,B 0,C 180,E1 33174.602,E2 33174.602} C_VEL
LIN {X 0,Y 726.657,Z 928.099,A -85,B 0,C 180,E1 33173.926,E2 33173.926} C_VEL
LIN {X 0,Y 727.127,Z 901.068,A -85,B 0,C 180,E1 33173.297,E2 33173.297} C_VEL
LIN {X 0,Y 727.454,Z 873.925,A -85,B 0,C 180,E1 33172.831,E2 33172.831} C_VEL
LIN {X 0,Y 728.661,Z 641.631,A -85,B 0,C 180,E1 33170.018,E2 33170.018} C_VEL
LIN {X 0,Y 729.769,Z 433.943,A -85,B 0,C 180,E1 33167.43,E2 33167.43} C_VEL
LIN {X 0,Y 729.775,Z 408.578,A -85,B 0,C 180,E1 33167.097,E2 33167.097} C_VEL
LIN {X 0,Y 722.646,Z 397.784,A -85,B 0,C 180,E1 33166.414,E2 33166.414} C_VEL
LIN {X 0,Y 720.221,Z 391.638,A -85,B 0,C 180,E1 33165.775,E2 33165.775} C_VEL
LIN {X 0,Y 720.196,Z 391.515,A -85,B 0,C 180,E1 33162.855,E2 33162.855} C_VEL
LIN {X 0,Y 720.199,Z 391.517,A -85,B 0,C 180,E1 33159.969,E2 33159.969} C_VEL
LIN {X 0,Y 720.208,Z 391.521,A -85,B 0,C 180,E1 33157.031,E2 33157.031} C_VEL
LIN {X 0,Y 720.212,Z 391.504,A -85,B 0,C 180,E1 33154.02,E2 33154.02} C_VEL
LIN {X 0,Y 720.22,Z 391.512,A -85,B 0,C 180,E1 33151.002,E2 33151.002} C_VEL
LIN {X 0,Y 720.219,Z 391.51,A -85,B 0,C 180,E1 33147.896,E2 33147.896} C_VEL
LIN {X 0,Y 720.214,Z 391.512,A -85,B 0,C 180,E1 33144.789,E2 33144.789} C_VEL
LIN {X 0,Y 720.215,Z 391.507,A -85,B 0,C 180,E1 33141.672,E2 33141.672} C_VEL
LIN {X 0,Y 720.213,Z 391.516,A -85,B 0,C 180,E1 33138.622,E2 33138.622} C_VEL
LIN {X 0,Y 720.22,Z 391.502,A -85,B 0,C 180,E1 33135.529,E2 33135.529} C_VEL
LIN {X 0,Y 720.203,Z 391.517,A -85,B 0,C 180,E1 33132.508,E2 33132.508} C_VEL
LIN {X 0,Y 720.209,Z 391.501,A -85,B 0,C 180,E1 33129.51,E2 33129.51} C_VEL
LIN {X 0,Y 720.187,Z 391.514,A -85,B 0,C 180,E1 33126.617,E2 33126.617} C_VEL
LIN {X 0,Y 720.208,Z 391.507,A -85,B 0,C 180,E1 33123.741,E2 33123.741} C_VEL
LIN {X 0,Y 720.199,Z 391.51,A -85,B 0,C 180,E1 33120.796,E2 33120.796} C_VEL
LIN {X 0,Y 720.209,Z 391.516,A -85,B 0,C 180,E1 33117.852,E2 33117.852} C_VEL
LIN {X 0,Y 720.212,Z 391.508,A -85,B 0,C 180,E1 33114.743,E2 33114.743} C_VEL
LIN {X 0,Y 720.196,Z 391.518,A -85,B 0,C 180,E1 33111.778,E2 33111.778} C_VEL
LIN {X 0,Y 720.214,Z 391.511,A -85,B 0,C 180,E1 33108.792,E2 33108.792} C_VEL
LIN {X 0,Y 720.179,Z 391.512,A -85,B 0,C 180,E1 33105.938,E2 33105.938} C_VEL
LIN {X 0,Y 720.216,Z 391.52,A -85,B 0,C 180,E1 33103.132,E2 33103.132} C_VEL
LIN {X 0,Y 720.197,Z 391.503,A -85,B 0,C 180,E1 33100.114,E2 33100.114} C_VEL
LIN {X 0,Y 720.196,Z 391.52,A -85,B 0,C 180,E1 33097.202,E2 33097.202} C_VEL
LIN {X 0,Y 720.214,Z 391.507,A -85,B 0,C 180,E1 33094.111,E2 33094.111} C_VEL
LIN {X 0,Y 720.175,Z 391.517,A -85,B 0,C 180,E1 33091.289,E2 33091.289} C_VEL
LIN {X 0,Y 720.217,Z 391.52,A -85,B 0,C 180,E1 33088.478,E2 33088.478} C_VEL
LIN {X 0,Y 720.185,Z 391.51,A -85,B 0,C 180,E1 33085.496,E2 33085.496} C_VEL
LIN {X 0,Y 720.193,Z 391.514,A -85,B 0,C 180,E1 33082.647,E2 33082.647} C_VEL
LIN {X 0,Y 720.208,Z 391.516,A -85,B 0,C 180,E1 33079.537,E2 33079.537} C_VEL
LIN {X 0,Y 720.174,Z 391.525,A -85,B 0,C 180,E1 33076.696,E2 33076.696} C_VEL
LIN {X 0,Y 720.223,Z 391.618,A -85,B 0,C 180,E1 33076.261,E2 33076.261} C_VEL
LIN {X 0,Y 721.486,Z 394.952,A -85,B 0,C 180,E1 33075.916,E2 33075.916} C_VEL
LIN {X 0,Y 727.467,Z 408.143,A -85,B 0,C 180,E1 33074.508,E2 33074.508} C_VEL
LIN {X 0,Y 727.217,Z 428.076,A -85,B 0,C 180,E1 33073.184,E2 33073.184} C_VEL
LIN {X 0,Y 729.916,Z 439.091,A -85,B 0,C 180,E1 33072.841,E2 33072.841} C_VEL
LIN {X 0,Y 728.762,Z 652.606,A -85,B 0,C 180,E1 33070.17,E2 33070.17} C_VEL
LIN {X 0,Y 727.645,Z 878.02,A -85,B 0,C 180,E1 33067.446,E2 33067.446} C_VEL
LIN {X 0,Y 727.385,Z 912.535,A -85,B 0,C 180,E1 33066.994,E2 33066.994} C_VEL
LIN {X 0,Y 726.974,Z 939.585,A -85,B 0,C 180,E1 33066.477,E2 33066.477} C_VEL
LIN {X 0,Y 726.533,Z 965.381,A -85,B 0,C 180,E1 33065.831,E2 33065.831} C_VEL
LIN {X 0,Y 725.977,Z 993.12,A -85,B 0,C 180,E1 33064.959,E2 33064.959} C_VEL
LIN {X 0,Y 725.376,Z 1016.909,A -85,B 0,C 180,E1 33064.06,E2 33064.06} C_VEL
LIN {X 0,Y 724.836,Z 1038.082,A -85,B 0,C 180,E1 33063.139,E2 33063.139} C_VEL
LIN {X 0,Y 724.294,Z 1060.25,A -85,B 0,C 180,E1 33062.045,E2 33062.045} C_VEL
LIN {X 0,Y 723.608,Z 1085.572,A -85,B 0,C 180,E1 33060.613,E2 33060.613} C_VEL
LIN {X 0,Y 723.05,Z 1105.189,A -85,B 0,C 180,E1 33059.358,E2 33059.358} C_VEL
LIN {X 0,Y 722.552,Z 1124.264,A -85,B 0,C 180,E1 33058.007,E2 33058.007} C_VEL
LIN {X 0,Y 721.99,Z 1146.721,A -85,B 0,C 180,E1 33056.22,E2 33056.22} C_VEL
LIN {X 0,Y 721.54,Z 1163.349,A -85,B 0,C 180,E1 33054.743,E2 33054.743} C_VEL
LIN {X 0,Y 721.211,Z 1180.064,A -85,B 0,C 180,E1 33053.103,E2 33053.103} C_VEL
LIN {X 0,Y 720.833,Z 1197.809,A -85,B 0,C 180,E1 33051.143,E2 33051.143} C_VEL
LIN {X 0,Y 720.569,Z 1211.426,A -85,B 0,C 180,E1 33049.456,E2 33049.456} C_VEL
LIN {X 0,Y 720.35,Z 1223.563,A -85,B 0,C 180,E1 33047.783,E2 33047.783} C_VEL
LIN {X 0,Y 720.208,Z 1236.855,A -85,B 0,C 180,E1 33045.71,E2 33045.71} C_VEL
LIN {X 0,Y 720.048,Z 1247.227,A -85,B 0,C 180,E1 33043.821,E2 33043.821} C_VEL
LIN {X 0,Y 719.992,Z 1255.335,A -85,B 0,C 180,E1 33042.127,E2 33042.127} C_VEL
LIN {X 0,Y 719.965,Z 1262.116,A -85,B 0,C 180,E1 33040.485,E2 33040.485} C_VEL
LIN {X 0,Y 719.92,Z 1268.038,A -85,B 0,C 180,E1 33038.791,E2 33038.791} C_VEL
LIN {X 0,Y 719.921,Z 1273.362,A -85,B 0,C 180,E1 33036.943,E2 33036.943} C_VEL
LIN {X 0,Y 719.91,Z 1277.922,A -85,B 0,C 180,E1 33034.784,E2 33034.784} C_VEL
LIN {X 0,Y 719.911,Z 1280.605,A -85,B 0,C 180,E1 33032.71,E2 33032.71} C_VEL
LIN {X 0,Y 719.87,Z 1281.736,A -85,B 0,C 180,E1 33030.959,E2 33030.959} C_VEL
LIN {X 0,Y 719.863,Z 1281.828,A -85,B 0,C 180,E1 33029.367,E2 33029.367} C_VEL
LIN {X 0,Y 719.906,Z 1280.949,A -85,B 0,C 180,E1 33027.695,E2 33027.695} C_VEL
LIN {X 0,Y 719.92,Z 1278.809,A -85,B 0,C 180,E1 33025.782,E2 33025.782} C_VEL
LIN {X 0,Y 719.928,Z 1274.743,A -85,B 0,C 180,E1 33023.625,E2 33023.625} C_VEL
LIN {X 0,Y 719.944,Z 1269.086,A -85,B 0,C 180,E1 33021.538,E2 33021.538} C_VEL
LIN {X 0,Y 719.969,Z 1263.062,A -85,B 0,C 180,E1 33019.765,E2 33019.765} C_VEL
LIN {X 0,Y 719.986,Z 1256.164,A -85,B 0,C 180,E1 33018.062,E2 33018.062} C_VEL
LIN {X 0,Y 720.024,Z 1248.907,A -85,B 0,C 180,E1 33016.513,E2 33016.513} C_VEL
LIN {X 0,Y 720.136,Z 1240.622,A -85,B 0,C 180,E1 33014.956,E2 33014.956} C_VEL
LIN {X 0,Y 720.273,Z 1230.725,A -85,B 0,C 180,E1 33013.305,E2 33013.305} C_VEL
LIN {X 0,Y 720.484,Z 1217.794,A -85,B 0,C 180,E1 33011.391,E2 33011.391} C_VEL
LIN {X 0,Y 720.737,Z 1202.137,A -85,B 0,C 180,E1 33009.372,E2 33009.372} C_VEL
LIN {X 0,Y 720.992,Z 1188.104,A -85,B 0,C 180,E1 33007.758,E2 33007.758} C_VEL
LIN {X 0,Y 721.366,Z 1172.466,A -85,B 0,C 180,E1 33006.13,E2 33006.13} C_VEL
LIN {X 0,Y 721.822,Z 1152.4,A -85,B 0,C 180,E1 33004.267,E2 33004.267} C_VEL
LIN {X 0,Y 722.268,Z 1135.012,A -85,B 0,C 180,E1 33002.822,E2 33002.822} C_VEL
LIN {X 0,Y 722.801,Z 1115.669,A -85,B 0,C 180,E1 33001.364,E2 33001.364} C_VEL
LIN {X 0,Y 723.4,Z 1092.25,A -85,B 0,C 180,E1 32999.799,E2 32999.799} C_VEL
LIN {X 0,Y 723.939,Z 1072.106,A -85,B 0,C 180,E1 32998.603,E2 32998.603} C_VEL
LIN {X 0,Y 724.543,Z 1050.966,A -85,B 0,C 180,E1 32997.48,E2 32997.48} C_VEL
LIN {X 0,Y 725.221,Z 1025.568,A -85,B 0,C 180,E1 32996.3,E2 32996.3} C_VEL
LIN {X 0,Y 725.728,Z 1002.283,A -85,B 0,C 180,E1 32995.373,E2 32995.373} C_VEL
LIN {X 0,Y 726.176,Z 981.293,A -85,B 0,C 180,E1 32994.651,E2 32994.651} C_VEL
LIN {X 0,Y 726.654,Z 958.232,A -85,B 0,C 180,E1 32993.974,E2 32993.974} C_VEL
LIN {X 0,Y 727.125,Z 931.204,A -85,B 0,C 180,E1 32993.344,E2 32993.344} C_VEL
LIN {X 0,Y 727.458,Z 903.913,A -85,B 0,C 180,E1 32992.876,E2 32992.876} C_VEL
LIN {X 0,Y 728.669,Z 670.202,A -85,B 0,C 180,E1 32990.045,E2 32990.045} C_VEL
LIN {X 0,Y 729.792,Z 460.648,A -85,B 0,C 180,E1 32987.433,E2 32987.433} C_VEL
LIN {X 0,Y 729.75,Z 437.642,A -85,B 0,C 180,E1 32987.128,E2 32987.128} C_VEL
LIN {X 0,Y 727.106,Z 427.36,A -85,B 0,C 180,E1 32986.786,E2 32986.786} C_VEL
LIN {X 0,Y 727.45,Z 407.616,A -85,B 0,C 180,E1 32985.454,E2 32985.454} C_VEL
LIN {X 0,Y 721.488,Z 394.948,A -85,B 0,C 180,E1 32984.084,E2 32984.084} C_VEL
LIN {X 0,Y 720.196,Z 391.524,A -85,B 0,C 180,E1 32983.71,E2 32983.71} C_VEL
LIN {X 0,Y 720.162,Z 391.509,A -85,B 0,C 180,E1 32980.958,E2 32980.958} C_VEL
LIN {X 0,Y 720.22,Z 391.514,A -85,B 0,C 180,E1 32978.088,E2 32978.088} C_VEL
LIN {X 0,Y 720.157,Z 391.519,A -85,B 0,C 180,E1 32975.184,E2 32975.184} C_VEL
LIN {X 0,Y 720.157,Z 391.517,A -85,B 0,C 180,E1 32972.596,E2 32972.596} C_VEL
LIN {X 0,Y 720.215,Z 391.511,A -85,B 0,C 180,E1 32969.62,E2 32969.62} C_VEL
LIN {X 0,Y 720.142,Z 391.519,A -85,B 0,C 180,E1 32966.913,E2 32966.913} C_VEL
LIN {X 0,Y 720.14,Z 391.514,A -85,B 0,C 180,E1 32964.442,E2 32964.442} C_VEL
LIN {X 0,Y 720.219,Z 391.516,A -85,B 0,C 180,E1 32961.557,E2 32961.557} C_VEL
LIN {X 0,Y 720.131,Z 391.521,A -85,B 0,C 180,E1 32958.769,E2 32958.769} C_VEL
LIN {X 0,Y 720.123,Z 391.52,A -85,B 0,C 180,E1 32956.396,E2 32956.396} C_VEL
LIN {X 0,Y 720.139,Z 391.513,A -85,B 0,C 180,E1 32953.971,E2 32953.971} C_VEL
LIN {X 0,Y 720.146,Z 391.519,A -85,B 0,C 180,E1 32950.885,E2 32950.885} C_VEL
LIN {X 0,Y 720.108,Z 391.517,A -85,B 0,C 180,E1 32948.383,E2 32948.383} C_VEL
LIN {X 0,Y 720.108,Z 391.524,A -85,B 0,C 180,E1 32946.138,E2 32946.138} C_VEL
LIN {X 0,Y 720.139,Z 391.518,A -85,B 0,C 180,E1 32943.662,E2 32943.662} C_VEL
LIN {X 0,Y 720.145,Z 391.522,A -85,B 0,C 180,E1 32940.557,E2 32940.557} C_VEL
LIN {X 0,Y 720.122,Z 391.516,A -85,B 0,C 180,E1 32938.09,E2 32938.09} C_VEL
LIN {X 0,Y 720.132,Z 391.516,A -85,B 0,C 180,E1 32935.7,E2 32935.7} C_VEL
LIN {X 0,Y 720.222,Z 391.514,A -85,B 0,C 180,E1 32932.822,E2 32932.822} C_VEL
LIN {X 0,Y 720.139,Z 391.514,A -85,B 0,C 180,E1 32930.005,E2 32930.005} C_VEL
LIN {X 0,Y 720.143,Z 391.521,A -85,B 0,C 180,E1 32927.572,E2 32927.572} C_VEL
LIN {X 0,Y 720.223,Z 391.509,A -85,B 0,C 180,E1 32924.788,E2 32924.788} C_VEL
LIN {X 0,Y 720.147,Z 391.516,A -85,B 0,C 180,E1 32923.493,E2 32923.493} C_VEL
LIN {X 0,Y 719.179,Z 391.648,A -85,B 0,C 180,E1 32922.88,E2 32922.88} C_VEL
LIN {X 0,Y 712.797,Z 392.444,A -85,B 0,C 180,E1 32921.163,E2 32921.163} C_VEL
LIN {X 0,Y 712.278,Z 392.5,A -85,B 0,C 180,E1 32920.717,E2 32920.717} C_VEL
LIN {X 0,Y 712.227,Z 392.505,A -85,B 0,C 180,E1 32917.812,E2 32917.812} C_VEL
LIN {X 0,Y 712.224,Z 392.506,A -85,B 0,C 180,E1 32915.18,E2 32915.18} C_VEL
LIN {X 0,Y 712.281,Z 392.505,A -85,B 0,C 180,E1 32912.221,E2 32912.221} C_VEL
LIN {X 0,Y 712.227,Z 392.495,A -85,B 0,C 180,E1 32909.362,E2 32909.362} C_VEL
LIN {X 0,Y 712.277,Z 392.504,A -85,B 0,C 180,E1 32906.517,E2 32906.517} C_VEL
LIN {X 0,Y 712.25,Z 392.505,A -85,B 0,C 180,E1 32903.471,E2 32903.471} C_VEL
LIN {X 0,Y 712.257,Z 392.501,A -85,B 0,C 180,E1 32900.614,E2 32900.614} C_VEL
LIN {X 0,Y 712.274,Z 392.502,A -85,B 0,C 180,E1 32897.528,E2 32897.528} C_VEL
LIN {X 0,Y 712.266,Z 392.631,A -85,B 0,C 180,E1 32894.685,E2 32894.685} C_VEL
LIN {X 0,Y 713.783,Z 396.278,A -85,B 0,C 180,E1 32894.289,E2 32894.289} C_VEL
LIN {X 0,Y 714.727,Z 398.592,A -85,B 0,C 180,E1 32894.079,E2 32894.079} C_VEL
LIN {X 0,Y 723.994,Z 412.719,A -85,B 0,C 180,E1 32893.183,E2 32893.183} C_VEL
LIN {X 0,Y 722.66,Z 619.69,A -85,B 0,C 180,E1 32890.573,E2 32890.573} C_VEL
LIN {X 0,Y 721.304,Z 844.871,A -85,B 0,C 180,E1 32887.827,E2 32887.827} C_VEL
LIN {X 0,Y 720.983,Z 882.129,A -85,B 0,C 180,E1 32887.341,E2 32887.341} C_VEL
LIN {X 0,Y 720.484,Z 909.348,A -85,B 0,C 180,E1 32886.82,E2 32886.82} C_VEL
LIN {X 0,Y 719.969,Z 934.955,A -85,B 0,C 180,E1 32886.177,E2 32886.177} C_VEL
LIN {X 0,Y 719.322,Z 962.268,A -85,B 0,C 180,E1 32885.317,E2 32885.317} C_VEL
LIN {X 0,Y 718.59,Z 986.705,A -85,B 0,C 180,E1 32884.391,E2 32884.391} C_VEL
LIN {X 0,Y 717.93,Z 1007.95,A -85,B 0,C 180,E1 32883.462,E2 32883.462} C_VEL
LIN {X 0,Y 717.241,Z 1030.355,A -85,B 0,C 180,E1 32882.348,E2 32882.348} C_VEL
LIN {X 0,Y 716.429,Z 1055.729,A -85,B 0,C 180,E1 32880.898,E2 32880.898} C_VEL
LIN {X 0,Y 715.758,Z 1075.325,A -85,B 0,C 180,E1 32879.632,E2 32879.632} C_VEL
LIN {X 0,Y 715.13,Z 1094.608,A -85,B 0,C 180,E1 32878.253,E2 32878.253} C_VEL
LIN {X 0,Y 714.454,Z 1116.886,A -85,B 0,C 180,E1 32876.459,E2 32876.459} C_VEL
LIN {X 0,Y 713.932,Z 1133.428,A -85,B 0,C 180,E1 32874.972,E2 32874.972} C_VEL
LIN {X 0,Y 713.489,Z 1150.549,A -85,B 0,C 180,E1 32873.273,E2 32873.273} C_VEL
LIN {X 0,Y 713.036,Z 1168.215,A -85,B 0,C 180,E1 32871.291,E2 32871.291} C_VEL
LIN {X 0,Y 712.726,Z 1181.148,A -85,B 0,C 180,E1 32869.671,E2 32869.671} C_VEL
LIN {X 0,Y 712.488,Z 1192.727,A -85,B 0,C 180,E1 32868.063,E2 32868.063} C_VEL
LIN {X 0,Y 712.277,Z 1205.137,A -85,B 0,C 180,E1 32866.133,E2 32866.133} C_VEL
LIN {X 0,Y 712.112,Z 1217.043,A -85,B 0,C 180,E1 32863.971,E2 32863.971} C_VEL
LIN {X 0,Y 712.019,Z 1225.402,A -85,B 0,C 180,E1 32862.204,E2 32862.204} C_VEL
LIN {X 0,Y 711.976,Z 1232.282,A -85,B 0,C 180,E1 32860.515,E2 32860.515} C_VEL
LIN {X 0,Y 711.92,Z 1238.177,A -85,B 0,C 180,E1 32858.802,E2 32858.802} C_VEL
LIN {X 0,Y 711.923,Z 1243.467,A -85,B 0,C 180,E1 32856.933,E2 32856.933} C_VEL
LIN {X 0,Y 711.911,Z 1247.99,A -85,B 0,C 180,E1 32854.749,E2 32854.749} C_VEL
LIN {X 0,Y 711.91,Z 1250.641,A -85,B 0,C 180,E1 32852.653,E2 32852.653} C_VEL
LIN {X 0,Y 711.87,Z 1251.748,A -85,B 0,C 180,E1 32850.882,E2 32850.882} C_VEL
LIN {X 0,Y 711.863,Z 1251.816,A -85,B 0,C 180,E1 32849.272,E2 32849.272} C_VEL
LIN {X 0,Y 711.902,Z 1250.913,A -85,B 0,C 180,E1 32847.582,E2 32847.582} C_VEL
LIN {X 0,Y 711.916,Z 1248.742,A -85,B 0,C 180,E1 32845.647,E2 32845.647} C_VEL
LIN {X 0,Y 711.925,Z 1244.643,A -85,B 0,C 180,E1 32843.464,E2 32843.464} C_VEL
LIN {X 0,Y 711.945,Z 1238.949,A -85,B 0,C 180,E1 32841.354,E2 32841.354} C_VEL
LIN {X 0,Y 711.978,Z 1232.897,A -85,B 0,C 180,E1 32839.559,E2 32839.559} C_VEL
LIN {X 0,Y 712.012,Z 1226.329,A -85,B 0,C 180,E1 32837.919,E2 32837.919} C_VEL
LIN {X 0,Y 712.059,Z 1219.051,A -85,B 0,C 180,E1 32836.343,E2 32836.343} C_VEL
LIN {X 0,Y 712.188,Z 1210.831,A -85,B 0,C 180,E1 32834.776,E2 32834.776} C_VEL
LIN {X 0,Y 712.366,Z 1200.957,A -85,B 0,C 180,E1 32833.106,E2 32833.106} C_VEL
LIN {X 0,Y 712.597,Z 1188.633,A -85,B 0,C 180,E1 32831.254,E2 32831.254} C_VEL
LIN {X 0,Y 712.929,Z 1172.446,A -85,B 0,C 180,E1 32829.128,E2 32829.128} C_VEL
LIN {X 0,Y 713.244,Z 1158.439,A -85,B 0,C 180,E1 32827.495,E2 32827.495} C_VEL
LIN {X 0,Y 713.663,Z 1143.68,A -85,B 0,C 180,E1 32825.936,E2 32825.936} C_VEL
LIN {X 0,Y 714.22,Z 1123.833,A -85,B 0,C 180,E1 32824.054,E2 32824.054} C_VEL
LIN {X 0,Y 714.778,Z 1106.016,A -85,B 0,C 180,E1 32822.55,E2 32822.55} C_VEL
LIN {X 0,Y 715.357,Z 1087.977,A -85,B 0,C 180,E1 32821.167,E2 32821.167} C_VEL
LIN {X 0,Y 716.125,Z 1064.284,A -85,B 0,C 180,E1 32819.544,E2 32819.544} C_VEL
LIN {X 0,Y 716.809,Z 1043.154,A -85,B 0,C 180,E1 32818.27,E2 32818.27} C_VEL
LIN {X 0,Y 717.492,Z 1022.762,A -85,B 0,C 180,E1 32817.171,E2 32817.171} C_VEL
LIN {X 0,Y 718.3,Z 998.572,A -85,B 0,C 180,E1 32816.018,E2 32816.018} C_VEL
LIN {X 0,Y 718.968,Z 972.731,A -85,B 0,C 180,E1 32814.972,E2 32814.972} C_VEL
LIN {X 0,Y 719.524,Z 951.069,A -85,B 0,C 180,E1 32814.222,E2 32814.222} C_VEL
LIN {X 0,Y 720.115,Z 927.962,A -85,B 0,C 180,E1 32813.543,E2 32813.543} C_VEL
LIN {X 0,Y 720.665,Z 900.902,A -85,B 0,C 180,E1 32812.91,E2 32812.91} C_VEL
LIN {X 0,Y 721.062,Z 873.848,A -85,B 0,C 180,E1 32812.445,E2 32812.445} C_VEL
LIN {X 0,Y 722.505,Z 643.793,A -85,B 0,C 180,E1 32809.635,E2 32809.635} C_VEL
LIN {X 0,Y 723.849,Z 435.99,A -85,B 0,C 180,E1 32807.026,E2 32807.026} C_VEL
LIN {X 0,Y 723.882,Z 412.408,A -85,B 0,C 180,E1 32806.714,E2 32806.714} C_VEL
LIN {X 0,Y 714.324,Z 397.848,A -85,B 0,C 180,E1 32805.782,E2 32805.782} C_VEL
LIN {X 0,Y 712.26,Z 392.512,A -85,B 0,C 180,E1 32805.191,E2 32805.191} C_VEL
LIN {X 0,Y 712.272,Z 392.501,A -85,B 0,C 180,E1 32802.255,E2 32802.255} C_VEL
LIN {X 0,Y 712.275,Z 392.508,A -85,B 0,C 180,E1 32799.203,E2 32799.203} C_VEL
LIN {X 0,Y 712.277,Z 392.501,A -85,B 0,C 180,E1 32796.128,E2 32796.128} C_VEL
LIN {X 0,Y 712.279,Z 392.507,A -85,B 0,C 180,E1 32793.062,E2 32793.062} C_VEL
LIN {X 0,Y 712.282,Z 392.489,A -85,B 0,C 180,E1 32789.983,E2 32789.983} C_VEL
LIN {X 0,Y 712.279,Z 392.504,A -85,B 0,C 180,E1 32786.874,E2 32786.874} C_VEL
LIN {X 0,Y 712.28,Z 392.498,A -85,B 0,C 180,E1 32783.755,E2 32783.755} C_VEL
LIN {X 0,Y 712.272,Z 392.499,A -85,B 0,C 180,E1 32780.718,E2 32780.718} C_VEL
LIN {X 0,Y 712.279,Z 392.499,A -85,B 0,C 180,E1 32777.567,E2 32777.567} C_VEL
LIN {X 0,Y 712.274,Z 392.496,A -85,B 0,C 180,E1 32774.47,E2 32774.47} C_VEL
LIN {X 0,Y 712.276,Z 392.499,A -85,B 0,C 180,E1 32771.334,E2 32771.334} C_VEL
LIN {X 0,Y 712.266,Z 392.495,A -85,B 0,C 180,E1 32768.314,E2 32768.314} C_VEL
LIN {X 0,Y 712.278,Z 392.498,A -85,B 0,C 180,E1 32765.235,E2 32765.235} C_VEL
LIN {X 0,Y 712.252,Z 392.493,A -85,B 0,C 180,E1 32762.253,E2 32762.253} C_VEL
LIN {X 0,Y 712.268,Z 392.503,A -85,B 0,C 180,E1 32759.357,E2 32759.357} C_VEL
LIN {X 0,Y 712.247,Z 392.488,A -85,B 0,C 180,E1 32756.459,E2 32756.459} C_VEL
LIN {X 0,Y 712.28,Z 392.509,A -85,B 0,C 180,E1 32753.552,E2 32753.552} C_VEL
LIN {X 0,Y 712.26,Z 392.488,A -85,B 0,C 180,E1 32750.465,E2 32750.465} C_VEL
LIN {X 0,Y 712.266,Z 392.51,A -85,B 0,C 180,E1 32747.515,E2 32747.515} C_VEL
LIN {X 0,Y 712.27,Z 392.493,A -85,B 0,C 180,E1 32744.364,E2 32744.364} C_VEL
LIN {X 0,Y 712.253,Z 392.509,A -85,B 0,C 180,E1 32741.417,E2 32741.417} C_VEL
LIN {X 0,Y 712.279,Z 392.5,A -85,B 0,C 180,E1 32738.42,E2 32738.42} C_VEL
LIN {X 0,Y 712.239,Z 392.502,A -85,B 0,C 180,E1 32735.623,E2 32735.623} C_VEL
LIN {X 0,Y 712.279,Z 392.51,A -85,B 0,C 180,E1 32732.765,E2 32732.765} C_VEL
LIN {X 0,Y 712.251,Z 392.496,A -85,B 0,C 180,E1 32729.698,E2 32729.698} C_VEL
LIN {X 0,Y 712.257,Z 392.505,A -85,B 0,C 180,E1 32726.793,E2 32726.793} C_VEL
LIN {X 0,Y 712.268,Z 392.5,A -85,B 0,C 180,E1 32723.672,E2 32723.672} C_VEL
LIN {X 0,Y 712.239,Z 392.51,A -85,B 0,C 180,E1 32720.801,E2 32720.801} C_VEL
LIN {X 0,Y 712.278,Z 392.511,A -85,B 0,C 180,E1 32717.956,E2 32717.956} C_VEL
LIN {X 0,Y 712.237,Z 392.545,A -85,B 0,C 180,E1 32716.867,E2 32716.867} C_VEL
LIN {X 0,Y 713.462,Z 395.862,A -85,B 0,C 180,E1 32716.518,E2 32716.518} C_VEL
LIN {X 0,Y 714.543,Z 398.031,A -85,B 0,C 180,E1 32716.269,E2 32716.269} C_VEL
LIN {X 0,Y 721.009,Z 412.127,A -85,B 0,C 180,E1 32714.733,E2 32714.733} C_VEL
LIN {X 0,Y 720.77,Z 428.038,A -85,B 0,C 180,E1 32713.667,E2 32713.667} C_VEL
LIN {X 0,Y 724.023,Z 441.264,A -85,B 0,C 180,E1 32713.246,E2 32713.246} C_VEL
LIN {X 0,Y 722.631,Z 653.887,A -85,B 0,C 180,E1 32710.566,E2 32710.566} C_VEL
LIN {X 0,Y 721.279,Z 879.154,A -85,B 0,C 180,E1 32707.821,E2 32707.821} C_VEL
LIN {X 0,Y 720.965,Z 912.978,A -85,B 0,C 180,E1 32707.372,E2 32707.372} C_VEL
LIN {X 0,Y 720.473,Z 939.955,A -85,B 0,C 180,E1 32706.851,E2 32706.851} C_VEL
LIN {X 0,Y 719.957,Z 965.421,A -85,B 0,C 180,E1 32706.209,E2 32706.209} C_VEL
LIN {X 0,Y 719.265,Z 993.701,A -85,B 0,C 180,E1 32705.311,E2 32705.311} C_VEL
LIN {X 0,Y 718.602,Z 1016.422,A -85,B 0,C 180,E1 32704.447,E2 32704.447} C_VEL
LIN {X 0,Y 717.942,Z 1037.635,A -85,B 0,C 180,E1 32703.521,E2 32703.521} C_VEL
LIN {X 0,Y 717.253,Z 1059.93,A -85,B 0,C 180,E1 32702.415,E2 32702.415} C_VEL
LIN {X 0,Y 716.467,Z 1084.839,A -85,B 0,C 180,E1 32700.998,E2 32700.998} C_VEL
LIN {X 0,Y 715.79,Z 1104.529,A -85,B 0,C 180,E1 32699.731,E2 32699.731} C_VEL
LIN {X 0,Y 715.191,Z 1122.809,A -85,B 0,C 180,E1 32698.431,E2 32698.431} C_VEL
LIN {X 0,Y 714.551,Z 1143.759,A -85,B 0,C 180,E1 32696.776,E2 32696.776} C_VEL
LIN {X 0,Y 713.97,Z 1162.418,A -85,B 0,C 180,E1 32695.111,E2 32695.111} C_VEL
LIN {X 0,Y 713.52,Z 1178.364,A -85,B 0,C 180,E1 32693.542,E2 32693.542} C_VEL
LIN {X 0,Y 713.061,Z 1197.1,A -85,B 0,C 180,E1 32691.471,E2 32691.471} C_VEL
LIN {X 0,Y 712.725,Z 1211.122,A -85,B 0,C 180,E1 32689.719,E2 32689.719} C_VEL
LIN {X 0,Y 712.48,Z 1222.982,A -85,B 0,C 180,E1 32688.071,E2 32688.071} C_VEL
LIN {X 0,Y 712.274,Z 1235.88,A -85,B 0,C 180,E1 32686.057,E2 32686.057} C_VEL
LIN {X 0,Y 712.103,Z 1247.228,A -85,B 0,C 180,E1 32683.979,E2 32683.979} C_VEL
LIN {X 0,Y 712.023,Z 1255.418,A -85,B 0,C 180,E1 32682.245,E2 32682.245} C_VEL
LIN {X 0,Y 711.974,Z 1262.423,A -85,B 0,C 180,E1 32680.523,E2 32680.523} C_VEL
LIN {X 0,Y 711.924,Z 1268.295,A -85,B 0,C 180,E1 32678.809,E2 32678.809} C_VEL
LIN {X 0,Y 711.923,Z 1273.557,A -85,B 0,C 180,E1 32676.941,E2 32676.941} C_VEL
LIN {X 0,Y 711.914,Z 1277.922,A -85,B 0,C 180,E1 32674.837,E2 32674.837} C_VEL
LIN {X 0,Y 711.912,Z 1280.606,A -85,B 0,C 180,E1 32672.741,E2 32672.741} C_VEL
LIN {X 0,Y 711.871,Z 1281.736,A -85,B 0,C 180,E1 32670.969,E2 32670.969} C_VEL
LIN {X 0,Y 711.863,Z 1281.828,A -85,B 0,C 180,E1 32669.36,E2 32669.36} C_VEL
LIN {X 0,Y 711.906,Z 1280.949,A -85,B 0,C 180,E1 32667.669,E2 32667.669} C_VEL
LIN {X 0,Y 711.919,Z 1278.809,A -85,B 0,C 180,E1 32665.735,E2 32665.735} C_VEL
LIN {X 0,Y 711.928,Z 1274.743,A -85,B 0,C 180,E1 32663.553,E2 32663.553} C_VEL
LIN {X 0,Y 711.947,Z 1269.087,A -85,B 0,C 180,E1 32661.443,E2 32661.443} C_VEL
LIN {X 0,Y 711.981,Z 1263.063,A -85,B 0,C 180,E1 32659.649,E2 32659.649} C_VEL
LIN {X 0,Y 712.009,Z 1256.166,A -85,B 0,C 180,E1 32657.926,E2 32657.926} C_VEL
LIN {X 0,Y 712.062,Z 1248.824,A -85,B 0,C 180,E1 32656.342,E2 32656.342} C_VEL
LIN {X 0,Y 712.194,Z 1240.624,A -85,B 0,C 180,E1 32654.784,E2 32654.784} C_VEL
LIN {X 0,Y 712.37,Z 1230.726,A -85,B 0,C 180,E1 32653.114,E2 32653.114} C_VEL
LIN {X 0,Y 712.638,Z 1217.214,A -85,B 0,C 180,E1 32651.093,E2 32651.093} C_VEL
LIN {X 0,Y 712.95,Z 1201.428,A -85,B 0,C 180,E1 32649.051,E2 32649.051} C_VEL
LIN {X 0,Y 713.276,Z 1187.326,A -85,B 0,C 180,E1 32647.417,E2 32647.417} C_VEL
LIN {X 0,Y 713.792,Z 1169.732,A -85,B 0,C 180,E1 32645.579,E2 32645.579} C_VEL
LIN {X 0,Y 714.31,Z 1150.876,A -85,B 0,C 180,E1 32643.842,E2 32643.842} C_VEL
LIN {X 0,Y 714.857,Z 1133.905,A -85,B 0,C 180,E1 32642.426,E2 32642.426} C_VEL
LIN {X 0,Y 715.558,Z 1112.595,A -85,B 0,C 180,E1 32640.818,E2 32640.818} C_VEL
LIN {X 0,Y 716.223,Z 1090.797,A -85,B 0,C 180,E1 32639.372,E2 32639.372} C_VEL
LIN {X 0,Y 716.87,Z 1071.726,A -85,B 0,C 180,E1 32638.235,E2 32638.235} C_VEL
LIN {X 0,Y 717.589,Z 1050.286,A -85,B 0,C 180,E1 32637.089,E2 32637.089} C_VEL
LIN {X 0,Y 718.379,Z 1024.454,A -85,B 0,C 180,E1 32635.887,E2 32635.887} C_VEL
LIN {X 0,Y 718.977,Z 1002.229,A -85,B 0,C 180,E1 32634.998,E2 32634.998} C_VEL
LIN {X 0,Y 719.538,Z 980.465,A -85,B 0,C 180,E1 32634.247,E2 32634.247} C_VEL
LIN {X 0,Y 720.134,Z 957.217,A -85,B 0,C 180,E1 32633.568,E2 32633.568} C_VEL
LIN {X 0,Y 720.67,Z 930.291,A -85,B 0,C 180,E1 32632.943,E2 32632.943} C_VEL
LIN {X 0,Y 721.073,Z 903.26,A -85,B 0,C 180,E1 32632.482,E2 32632.482} C_VEL
LIN {X 0,Y 722.522,Z 670.949,A -85,B 0,C 180,E1 32629.645,E2 32629.645} C_VEL
LIN {X 0,Y 723.884,Z 461.411,A -85,B 0,C 180,E1 32627.012,E2 32627.012} C_VEL
LIN {X 0,Y 723.866,Z 439.884,A -85,B 0,C 180,E1 32626.724,E2 32626.724} C_VEL
LIN {X 0,Y 720.671,Z 427.188,A -85,B 0,C 180,E1 32626.291,E2 32626.291} C_VEL
LIN {X 0,Y 720.954,Z 411.849,A -85,B 0,C 180,E1 32625.243,E2 32625.243} C_VEL
LIN {X 0,Y 715.23,Z 399.568,A -85,B 0,C 180,E1 32623.901,E2 32623.901} C_VEL
LIN {X 0,Y 713.88,Z 396.456,A -85,B 0,C 180,E1 32623.56,E2 32623.56} C_VEL
LIN {X 0,Y 712.32,Z 393.099,A -85,B 0,C 180,E1 32623.181,E2 32623.181} C_VEL
LIN {X 0,Y 712.225,Z 392.514,A -85,B 0,C 180,E1 32623.12,E2 32623.12} C_VEL
LIN {X 0,Y 712.282,Z 392.492,A -85,B 0,C 180,E1 32620.327,E2 32620.327} C_VEL
LIN {X 0,Y 712.225,Z 392.504,A -85,B 0,C 180,E1 32617.336,E2 32617.336} C_VEL
LIN {X 0,Y 712.217,Z 392.505,A -85,B 0,C 180,E1 32614.75,E2 32614.75} C_VEL
LIN {X 0,Y 712.284,Z 392.507,A -85,B 0,C 180,E1 32611.859,E2 32611.859} C_VEL
LIN {X 0,Y 712.207,Z 392.507,A -85,B 0,C 180,E1 32609.01,E2 32609.01} C_VEL
LIN {X 0,Y 712.205,Z 392.507,A -85,B 0,C 180,E1 32606.516,E2 32606.516} C_VEL
LIN {X 0,Y 712.285,Z 392.502,A -85,B 0,C 180,E1 32603.671,E2 32603.671} C_VEL
LIN {X 0,Y 712.196,Z 392.5,A -85,B 0,C 180,E1 32600.806,E2 32600.806} C_VEL
LIN {X 0,Y 712.189,Z 392.509,A -85,B 0,C 180,E1 32598.385,E2 32598.385} C_VEL
LIN {X 0,Y 712.256,Z 392.505,A -85,B 0,C 180,E1 32595.654,E2 32595.654} C_VEL
LIN {X 0,Y 712.19,Z 392.512,A -85,B 0,C 180,E1 32592.734,E2 32592.734} C_VEL
LIN {X 0,Y 712.172,Z 392.507,A -85,B 0,C 180,E1 32590.353,E2 32590.353} C_VEL
LIN {X 0,Y 712.176,Z 392.505,A -85,B 0,C 180,E1 32587.99,E2 32587.99} C_VEL
LIN {X 0,Y 712.268,Z 392.507,A -85,B 0,C 180,E1 32585.155,E2 32585.155} C_VEL
LIN {X 0,Y 712.18,Z 392.504,A -85,B 0,C 180,E1 32582.333,E2 32582.333} C_VEL
LIN {X 0,Y 712.181,Z 392.511,A -85,B 0,C 180,E1 32580,E2 32580} C_VEL
LIN {X 0,Y 712.21,Z 392.505,A -85,B 0,C 180,E1 32577.506,E2 32577.506} C_VEL
LIN {X 0,Y 712.212,Z 392.509,A -85,B 0,C 180,E1 32574.36,E2 32574.36} C_VEL
LIN {X 0,Y 712.193,Z 392.503,A -85,B 0,C 180,E1 32571.848,E2 32571.848} C_VEL
LIN {X 0,Y 712.224,Z 392.505,A -85,B 0,C 180,E1 32569.298,E2 32569.298} C_VEL
LIN {X 0,Y 712.23,Z 392.499,A -85,B 0,C 180,E1 32566.192,E2 32566.192} C_VEL
LIN {X 0,Y 712.206,Z 392.504,A -85,B 0,C 180,E1 32563.609,E2 32563.609} C_VEL
LIN {X 0,Y 712.259,Z 392.508,A -85,B 0,C 180,E1 32560.908,E2 32560.908} C_VEL
LIN {X 0,Y 712.278,Z 392.5,A -85,B 0,C 180,E1 32560.717,E2 32560.717} C_VEL
LIN {X 0,Y 711.308,Z 392.612,A -85,B 0,C 180,E1 32560.097,E2 32560.097} C_VEL
LIN {X 0,Y 704.862,Z 393.428,A -85,B 0,C 180,E1 32558.362,E2 32558.362} C_VEL
LIN {X 0,Y 704.298,Z 393.493,A -85,B 0,C 180,E1 32557.911,E2 32557.911} C_VEL
LIN {X 0,Y 704.283,Z 393.495,A -85,B 0,C 180,E1 32555.24,E2 32555.24} C_VEL
LIN {X 0,Y 704.341,Z 393.496,A -85,B 0,C 180,E1 32552.34,E2 32552.34} C_VEL
LIN {X 0,Y 704.291,Z 393.481,A -85,B 0,C 180,E1 32549.452,E2 32549.452} C_VEL
LIN {X 0,Y 704.322,Z 393.498,A -85,B 0,C 180,E1 32546.674,E2 32546.674} C_VEL
LIN {X 0,Y 704.322,Z 393.493,A -85,B 0,C 180,E1 32543.594,E2 32543.594} C_VEL
LIN {X 0,Y 704.313,Z 393.488,A -85,B 0,C 180,E1 32540.679,E2 32540.679} C_VEL
LIN {X 0,Y 704.339,Z 393.491,A -85,B 0,C 180,E1 32537.69,E2 32537.69} C_VEL
LIN {X 0,Y 704.351,Z 393.722,A -85,B 0,C 180,E1 32535.241,E2 32535.241} C_VEL
LIN {X 0,Y 705.697,Z 397.106,A -85,B 0,C 180,E1 32534.87,E2 32534.87} C_VEL
LIN {X 0,Y 706.582,Z 398.879,A -85,B 0,C 180,E1 32534.719,E2 32534.719} C_VEL
LIN {X 0,Y 718.125,Z 416.335,A -85,B 0,C 180,E1 32533.576,E2 32533.576} C_VEL
LIN {X 0,Y 716.559,Z 622.11,A -85,B 0,C 180,E1 32530.961,E2 32530.961} C_VEL
LIN {X 0,Y 714.968,Z 846.796,A -85,B 0,C 180,E1 32528.199,E2 32528.199} C_VEL
LIN {X 0,Y 714.597,Z 882.516,A -85,B 0,C 180,E1 32527.726,E2 32527.726} C_VEL
LIN {X 0,Y 714.019,Z 909.765,A -85,B 0,C 180,E1 32527.2,E2 32527.2} C_VEL
LIN {X 0,Y 713.426,Z 934.91,A -85,B 0,C 180,E1 32526.564,E2 32526.564} C_VEL
LIN {X 0,Y 712.633,Z 963.059,A -85,B 0,C 180,E1 32525.669,E2 32525.669} C_VEL
LIN {X 0,Y 711.828,Z 986.723,A -85,B 0,C 180,E1 32524.764,E2 32524.764} C_VEL
LIN {X 0,Y 711.063,Z 1007.894,A -85,B 0,C 180,E1 32523.832,E2 32523.832} C_VEL
LIN {X 0,Y 710.23,Z 1030.149,A -85,B 0,C 180,E1 32522.719,E2 32522.719} C_VEL
LIN {X 0,Y 709.308,Z 1055.002,A -85,B 0,C 180,E1 32521.29,E2 32521.29} C_VEL
LIN {X 0,Y 708.523,Z 1074.673,A -85,B 0,C 180,E1 32520.012,E2 32520.012} C_VEL
LIN {X 0,Y 707.801,Z 1093.494,A -85,B 0,C 180,E1 32518.658,E2 32518.658} C_VEL
LIN {X 0,Y 706.97,Z 1115.804,A -85,B 0,C 180,E1 32516.858,E2 32516.858} C_VEL
LIN {X 0,Y 706.363,Z 1132.969,A -85,B 0,C 180,E1 32515.303,E2 32515.303} C_VEL
LIN {X 0,Y 705.804,Z 1149.708,A -85,B 0,C 180,E1 32513.63,E2 32513.63} C_VEL
LIN {X 0,Y 705.275,Z 1167.512,A -85,B 0,C 180,E1 32511.625,E2 32511.625} C_VEL
LIN {X 0,Y 704.883,Z 1181.154,A -85,B 0,C 180,E1 32509.899,E2 32509.899} C_VEL
LIN {X 0,Y 704.604,Z 1193.315,A -85,B 0,C 180,E1 32508.187,E2 32508.187} C_VEL
LIN {X 0,Y 704.333,Z 1206.826,A -85,B 0,C 180,E1 32506.035,E2 32506.035} C_VEL
LIN {X 0,Y 704.156,Z 1217.458,A -85,B 0,C 180,E1 32504.048,E2 32504.048} C_VEL
LIN {X 0,Y 704.047,Z 1225.667,A -85,B 0,C 180,E1 32502.284,E2 32502.284} C_VEL
LIN {X 0,Y 703.985,Z 1232.345,A -85,B 0,C 180,E1 32500.62,E2 32500.62} C_VEL
LIN {X 0,Y 703.919,Z 1238.179,A -85,B 0,C 180,E1 32498.903,E2 32498.903} C_VEL
LIN {X 0,Y 703.929,Z 1243.468,A -85,B 0,C 180,E1 32497.013,E2 32497.013} C_VEL
LIN {X 0,Y 703.913,Z 1247.99,A -85,B 0,C 180,E1 32494.803,E2 32494.803} C_VEL
LIN {X 0,Y 703.911,Z 1250.642,A -85,B 0,C 180,E1 32492.683,E2 32492.683} C_VEL
LIN {X 0,Y 703.871,Z 1251.748,A -85,B 0,C 180,E1 32490.892,E2 32490.892} C_VEL
LIN {X 0,Y 703.863,Z 1251.816,A -85,B 0,C 180,E1 32489.264,E2 32489.264} C_VEL
LIN {X 0,Y 703.902,Z 1250.913,A -85,B 0,C 180,E1 32487.554,E2 32487.554} C_VEL
LIN {X 0,Y 703.914,Z 1248.741,A -85,B 0,C 180,E1 32485.597,E2 32485.597} C_VEL
LIN {X 0,Y 703.923,Z 1244.642,A -85,B 0,C 180,E1 32483.39,E2 32483.39} C_VEL
LIN {X 0,Y 703.942,Z 1238.948,A -85,B 0,C 180,E1 32481.255,E2 32481.255} C_VEL
LIN {X 0,Y 703.984,Z 1232.896,A -85,B 0,C 180,E1 32479.439,E2 32479.439} C_VEL
LIN {X 0,Y 704.038,Z 1226.328,A -85,B 0,C 180,E1 32477.78,E2 32477.78} C_VEL
LIN {X 0,Y 704.113,Z 1218.681,A -85,B 0,C 180,E1 32476.111,E2 32476.111} C_VEL
LIN {X 0,Y 704.284,Z 1209.899,A -85,B 0,C 180,E1 32474.432,E2 32474.432} C_VEL
LIN {X 0,Y 704.488,Z 1198.342,A -85,B 0,C 180,E1 32472.486,E2 32472.486} C_VEL
LIN {X 0,Y 704.837,Z 1183.701,A -85,B 0,C 180,E1 32470.351,E2 32470.351} C_VEL
LIN {X 0,Y 705.192,Z 1170.311,A -85,B 0,C 180,E1 32468.627,E2 32468.627} C_VEL
LIN {X 0,Y 705.605,Z 1156.095,A -85,B 0,C 180,E1 32466.974,E2 32466.974} C_VEL
LIN {X 0,Y 706.206,Z 1136.896,A -85,B 0,C 180,E1 32464.979,E2 32464.979} C_VEL
LIN {X 0,Y 706.842,Z 1119.575,A -85,B 0,C 180,E1 32463.383,E2 32463.383} C_VEL
LIN {X 0,Y 707.517,Z 1101.458,A -85,B 0,C 180,E1 32461.868,E2 32461.868} C_VEL
LIN {X 0,Y 708.369,Z 1078.482,A -85,B 0,C 180,E1 32460.159,E2 32460.159} C_VEL
LIN {X 0,Y 709.124,Z 1059.18,A -85,B 0,C 180,E1 32458.881,E2 32458.881} C_VEL
LIN {X 0,Y 709.886,Z 1039.934,A -85,B 0,C 180,E1 32457.733,E2 32457.733} C_VEL
LIN {X 0,Y 710.833,Z 1015.518,A -85,B 0,C 180,E1 32456.438,E2 32456.438} C_VEL
LIN {X 0,Y 711.656,Z 990.807,A -85,B 0,C 180,E1 32455.315,E2 32455.315} C_VEL
LIN {X 0,Y 712.371,Z 969.403,A -85,B 0,C 180,E1 32454.47,E2 32454.47} C_VEL
LIN {X 0,Y 713.046,Z 947.214,A -85,B 0,C 180,E1 32453.716,E2 32453.716} C_VEL
LIN {X 0,Y 713.773,Z 921.486,A -85,B 0,C 180,E1 32452.986,E2 32452.986} C_VEL
LIN {X 0,Y 714.363,Z 894.397,A -85,B 0,C 180,E1 32452.395,E2 32452.395} C_VEL
LIN {X 0,Y 714.769,Z 869.013,A -85,B 0,C 180,E1 32451.986,E2 32451.986} C_VEL
LIN {X 0,Y 716.419,Z 640.512,A -85,B 0,C 180,E1 32449.179,E2 32449.179} C_VEL
LIN {X 0,Y 717.996,Z 433.749,A -85,B 0,C 180,E1 32446.559,E2 32446.559} C_VEL
LIN {X 0,Y 717.963,Z 415.871,A -85,B 0,C 180,E1 32446.315,E2 32446.315} C_VEL
LIN {X 0,Y 706.112,Z 397.87,A -85,B 0,C 180,E1 32445.132,E2 32445.132} C_VEL
LIN {X 0,Y 704.524,Z 394.52,A -85,B 0,C 180,E1 32444.745,E2 32444.745} C_VEL
LIN {X 0,Y 704.332,Z 393.496,A -85,B 0,C 180,E1 32444.646,E2 32444.646} C_VEL
LIN {X 0,Y 704.329,Z 393.5,A -85,B 0,C 180,E1 32441.636,E2 32441.636} C_VEL
LIN {X 0,Y 704.32,Z 393.497,A -85,B 0,C 180,E1 32438.761,E2 32438.761} C_VEL
LIN {X 0,Y 704.322,Z 393.494,A -85,B 0,C 180,E1 32435.842,E2 32435.842} C_VEL
LIN {X 0,Y 704.334,Z 393.499,A -85,B 0,C 180,E1 32432.937,E2 32432.937} C_VEL
LIN {X 0,Y 704.335,Z 393.478,A -85,B 0,C 180,E1 32429.887,E2 32429.887} C_VEL
LIN {X 0,Y 704.341,Z 393.49,A -85,B 0,C 180,E1 32426.836,E2 32426.836} C_VEL
LIN {X 0,Y 704.336,Z 393.488,A -85,B 0,C 180,E1 32423.688,E2 32423.688} C_VEL
LIN {X 0,Y 704.337,Z 393.484,A -85,B 0,C 180,E1 32420.614,E2 32420.614} C_VEL
LIN {X 0,Y 704.338,Z 393.488,A -85,B 0,C 180,E1 32417.515,E2 32417.515} C_VEL
LIN {X 0,Y 704.334,Z 393.483,A -85,B 0,C 180,E1 32414.469,E2 32414.469} C_VEL
LIN {X 0,Y 704.335,Z 393.488,A -85,B 0,C 180,E1 32411.298,E2 32411.298} C_VEL
LIN {X 0,Y 704.332,Z 393.482,A -85,B 0,C 180,E1 32408.244,E2 32408.244} C_VEL
LIN {X 0,Y 704.339,Z 393.487,A -85,B 0,C 180,E1 32405.131,E2 32405.131} C_VEL
LIN {X 0,Y 704.322,Z 393.481,A -85,B 0,C 180,E1 32402.115,E2 32402.115} C_VEL
LIN {X 0,Y 704.341,Z 393.487,A -85,B 0,C 180,E1 32399.024,E2 32399.024} C_VEL
LIN {X 0,Y 704.308,Z 393.479,A -85,B 0,C 180,E1 32396.093,E2 32396.093} C_VEL
LIN {X 0,Y 704.331,Z 393.491,A -85,B 0,C 180,E1 32393.151,E2 32393.151} C_VEL
LIN {X 0,Y 704.309,Z 393.477,A -85,B 0,C 180,E1 32390.274,E2 32390.274} C_VEL
LIN {X 0,Y 704.339,Z 393.498,A -85,B 0,C 180,E1 32387.372,E2 32387.372} C_VEL
LIN {X 0,Y 704.321,Z 393.482,A -85,B 0,C 180,E1 32384.266,E2 32384.266} C_VEL
LIN {X 0,Y 704.326,Z 393.497,A -85,B 0,C 180,E1 32381.286,E2 32381.286} C_VEL
LIN {X 0,Y 704.332,Z 393.488,A -85,B 0,C 180,E1 32378.164,E2 32378.164} C_VEL
LIN {X 0,Y 704.309,Z 393.491,A -85,B 0,C 180,E1 32375.241,E2 32375.241} C_VEL
LIN {X 0,Y 704.342,Z 393.49,A -85,B 0,C 180,E1 32372.181,E2 32372.181} C_VEL
LIN {X 0,Y 704.298,Z 393.488,A -85,B 0,C 180,E1 32369.356,E2 32369.356} C_VEL
LIN {X 0,Y 704.338,Z 393.485,A -85,B 0,C 180,E1 32366.48,E2 32366.48} C_VEL
LIN {X 0,Y 704.31,Z 393.491,A -85,B 0,C 180,E1 32363.471,E2 32363.471} C_VEL
LIN {X 0,Y 704.313,Z 393.502,A -85,B 0,C 180,E1 32360.61,E2 32360.61} C_VEL
LIN {X 0,Y 704.34,Z 393.573,A -85,B 0,C 180,E1 32357.48,E2 32357.48} C_VEL
LIN {X 0,Y 705.628,Z 397.018,A -85,B 0,C 180,E1 32357.107,E2 32357.107} C_VEL
LIN {X 0,Y 712.029,Z 410.521,A -85,B 0,C 180,E1 32355.57,E2 32355.57} C_VEL
LIN {X 0,Y 714.542,Z 416.09,A -85,B 0,C 180,E1 32354.966,E2 32354.966} C_VEL
LIN {X 0,Y 714.388,Z 428.178,A -85,B 0,C 180,E1 32354.156,E2 32354.156} C_VEL
LIN {X 0,Y 718.168,Z 443.3,A -85,B 0,C 180,E1 32353.659,E2 32353.659} C_VEL
LIN {X 0,Y 716.53,Z 655.792,A -85,B 0,C 180,E1 32350.96,E2 32350.96} C_VEL
LIN {X 0,Y 714.937,Z 881.273,A -85,B 0,C 180,E1 32348.19,E2 32348.19} C_VEL
LIN {X 0,Y 714.564,Z 913.911,A -85,B 0,C 180,E1 32347.748,E2 32347.748} C_VEL
LIN {X 0,Y 713.998,Z 940.628,A -85,B 0,C 180,E1 32347.225,E2 32347.225} C_VEL
LIN {X 0,Y 713.396,Z 966.007,A -85,B 0,C 180,E1 32346.578,E2 32346.578} C_VEL
LIN {X 0,Y 712.603,Z 993.799,A -85,B 0,C 180,E1 32345.688,E2 32345.688} C_VEL
LIN {X 0,Y 711.841,Z 1016.425,A -85,B 0,C 180,E1 32344.821,E2 32344.821} C_VEL
LIN {X 0,Y 711.073,Z 1037.639,A -85,B 0,C 180,E1 32343.888,E2 32343.888} C_VEL
LIN {X 0,Y 710.259,Z 1059.22,A -85,B 0,C 180,E1 32342.812,E2 32342.812} C_VEL
LIN {X 0,Y 709.316,Z 1084.837,A -85,B 0,C 180,E1 32341.345,E2 32341.345} C_VEL
LIN {X 0,Y 708.533,Z 1104.531,A -85,B 0,C 180,E1 32340.067,E2 32340.067} C_VEL
LIN {X 0,Y 707.826,Z 1122.826,A -85,B 0,C 180,E1 32338.753,E2 32338.753} C_VEL
LIN {X 0,Y 707.03,Z 1144.182,A -85,B 0,C 180,E1 32337.046,E2 32337.046} C_VEL
LIN {X 0,Y 706.388,Z 1162.419,A -85,B 0,C 180,E1 32335.4,E2 32335.4} C_VEL
LIN {X 0,Y 705.829,Z 1178.751,A -85,B 0,C 180,E1 32333.774,E2 32333.774} C_VEL
LIN {X 0,Y 705.286,Z 1197.102,A -85,B 0,C 180,E1 32331.72,E2 32331.72} C_VEL
LIN {X 0,Y 704.892,Z 1210.785,A -85,B 0,C 180,E1 32329.993,E2 32329.993} C_VEL
LIN {X 0,Y 704.615,Z 1222.984,A -85,B 0,C 180,E1 32328.28,E2 32328.28} C_VEL
LIN {X 0,Y 704.341,Z 1236.387,A -85,B 0,C 180,E1 32326.158,E2 32326.158} C_VEL
LIN {X 0,Y 704.157,Z 1247.401,A -85,B 0,C 180,E1 32324.105,E2 32324.105} C_VEL
LIN {X 0,Y 704.058,Z 1255.42,A -85,B 0,C 180,E1 32322.386,E2 32322.386} C_VEL
LIN {X 0,Y 703.983,Z 1262.424,A -85,B 0,C 180,E1 32320.643,E2 32320.643} C_VEL
LIN {X 0,Y 703.915,Z 1268.04,A -85,B 0,C 180,E1 32318.993,E2 32318.993} C_VEL
LIN {X 0,Y 703.934,Z 1273.362,A -85,B 0,C 180,E1 32317.102,E2 32317.102} C_VEL
LIN {X 0,Y 703.916,Z 1277.922,A -85,B 0,C 180,E1 32314.893,E2 32314.893} C_VEL
LIN {X 0,Y 703.913,Z 1280.606,A -85,B 0,C 180,E1 32312.772,E2 32312.772} C_VEL
LIN {X 0,Y 703.872,Z 1281.736,A -85,B 0,C 180,E1 32310.98,E2 32310.98} C_VEL
LIN {X 0,Y 703.863,Z 1281.828,A -85,B 0,C 180,E1 32309.353,E2 32309.353} C_VEL
LIN {X 0,Y 703.906,Z 1280.949,A -85,B 0,C 180,E1 32307.643,E2 32307.643} C_VEL
LIN {X 0,Y 703.917,Z 1278.809,A -85,B 0,C 180,E1 32305.686,E2 32305.686} C_VEL
LIN {X 0,Y 703.928,Z 1274.743,A -85,B 0,C 180,E1 32303.479,E2 32303.479} C_VEL
LIN {X 0,Y 703.946,Z 1269.083,A -85,B 0,C 180,E1 32301.343,E2 32301.343} C_VEL
LIN {X 0,Y 703.989,Z 1263.063,A -85,B 0,C 180,E1 32299.53,E2 32299.53} C_VEL
LIN {X 0,Y 704.038,Z 1256.167,A -85,B 0,C 180,E1 32297.788,E2 32297.788} C_VEL
LIN {X 0,Y 704.117,Z 1248.499,A -85,B 0,C 180,E1 32296.119,E2 32296.119} C_VEL
LIN {X 0,Y 704.292,Z 1239.695,A -85,B 0,C 180,E1 32294.44,E2 32294.44} C_VEL
LIN {X 0,Y 704.504,Z 1227.593,A -85,B 0,C 180,E1 32292.409,E2 32292.409} C_VEL
LIN {X 0,Y 704.843,Z 1213.424,A -85,B 0,C 180,E1 32290.359,E2 32290.359} C_VEL
LIN {X 0,Y 705.203,Z 1200.009,A -85,B 0,C 180,E1 32288.635,E2 32288.635} C_VEL
LIN {X 0,Y 705.66,Z 1184.754,A -85,B 0,C 180,E1 32286.869,E2 32286.869} C_VEL
LIN {X 0,Y 706.267,Z 1165.3,A -85,B 0,C 180,E1 32284.873,E2 32284.873} C_VEL
LIN {X 0,Y 706.868,Z 1148.845,A -85,B 0,C 180,E1 32283.364,E2 32283.364} C_VEL
LIN {X 0,Y 707.575,Z 1130.023,A -85,B 0,C 180,E1 32281.797,E2 32281.797} C_VEL
LIN {X 0,Y 708.389,Z 1107.961,A -85,B 0,C 180,E1 32280.168,E2 32280.168} C_VEL
LIN {X 0,Y 709.15,Z 1088.615,A -85,B 0,C 180,E1 32278.891,E2 32278.891} C_VEL
LIN {X 0,Y 709.944,Z 1068.508,A -85,B 0,C 180,E1 32277.697,E2 32277.697} C_VEL
LIN {X 0,Y 710.886,Z 1042.79,A -85,B 0,C 180,E1 32276.353,E2 32276.353} C_VEL
LIN {X 0,Y 711.688,Z 1019.986,A -85,B 0,C 180,E1 32275.326,E2 32275.326} C_VEL
LIN {X 0,Y 712.41,Z 998.477,A -85,B 0,C 180,E1 32274.482,E2 32274.482} C_VEL
LIN {X 0,Y 713.127,Z 974.669,A -85,B 0,C 180,E1 32273.68,E2 32273.68} C_VEL
LIN {X 0,Y 713.848,Z 948.007,A -85,B 0,C 180,E1 32272.947,E2 32272.947} C_VEL
LIN {X 0,Y 714.398,Z 922.292,A -85,B 0,C 180,E1 32272.401,E2 32272.401} C_VEL
LIN {X 0,Y 714.805,Z 896.296,A -85,B 0,C 180,E1 32271.995,E2 32271.995} C_VEL
LIN {X 0,Y 716.433,Z 668.675,A -85,B 0,C 180,E1 32269.201,E2 32269.201} C_VEL
LIN {X 0,Y 718.036,Z 459.376,A -85,B 0,C 180,E1 32266.548,E2 32266.548} C_VEL
LIN {X 0,Y 718.023,Z 442.084,A -85,B 0,C 180,E1 32266.314,E2 32266.314} C_VEL
LIN {X 0,Y 714.251,Z 427.36,A -85,B 0,C 180,E1 32265.809,E2 32265.809} C_VEL
LIN {X 0,Y 714.448,Z 415.906,A -85,B 0,C 180,E1 32265.013,E2 32265.013} C_VEL
LIN {X 0,Y 708.016,Z 401.763,A -85,B 0,C 180,E1 32263.453,E2 32263.453} C_VEL
LIN {X 0,Y 704.518,Z 394.533,A -85,B 0,C 180,E1 32262.609,E2 32262.609} C_VEL
LIN {X 0,Y 704.329,Z 393.499,A -85,B 0,C 180,E1 32262.512,E2 32262.512} C_VEL
LIN {X 0,Y 704.297,Z 393.503,A -85,B 0,C 180,E1 32259.448,E2 32259.448} C_VEL
LIN {X 0,Y 704.281,Z 393.493,A -85,B 0,C 180,E1 32256.808,E2 32256.808} C_VEL
LIN {X 0,Y 704.345,Z 393.484,A -85,B 0,C 180,E1 32253.865,E2 32253.865} C_VEL
LIN {X 0,Y 704.271,Z 393.495,A -85,B 0,C 180,E1 32251.022,E2 32251.022} C_VEL
LIN {X 0,Y 704.273,Z 393.494,A -85,B 0,C 180,E1 32248.492,E2 32248.492} C_VEL
LIN {X 0,Y 704.336,Z 393.485,A -85,B 0,C 180,E1 32245.567,E2 32245.567} C_VEL
LIN {X 0,Y 704.258,Z 393.5,A -85,B 0,C 180,E1 32242.805,E2 32242.805} C_VEL
LIN {X 0,Y 704.256,Z 393.487,A -85,B 0,C 180,E1 32240.356,E2 32240.356} C_VEL
LIN {X 0,Y 704.337,Z 393.5,A -85,B 0,C 180,E1 32237.43,E2 32237.43} C_VEL
LIN {X 0,Y 704.245,Z 393.489,A -85,B 0,C 180,E1 32234.639,E2 32234.639} C_VEL
LIN {X 0,Y 704.238,Z 393.501,A -85,B 0,C 180,E1 32232.297,E2 32232.297} C_VEL
LIN {X 0,Y 704.271,Z 393.495,A -85,B 0,C 180,E1 32229.727,E2 32229.727} C_VEL
LIN {X 0,Y 704.253,Z 393.502,A -85,B 0,C 180,E1 32226.686,E2 32226.686} C_VEL
LIN {X 0,Y 704.234,Z 393.494,A -85,B 0,C 180,E1 32224.234,E2 32224.234} C_VEL
LIN {X 0,Y 704.247,Z 393.493,A -85,B 0,C 180,E1 32221.79,E2 32221.79} C_VEL
LIN {X 0,Y 704.322,Z 393.491,A -85,B 0,C 180,E1 32218.861,E2 32218.861} C_VEL
LIN {X 0,Y 704.249,Z 393.491,A -85,B 0,C 180,E1 32216.092,E2 32216.092} C_VEL
LIN {X 0,Y 704.26,Z 393.5,A -85,B 0,C 180,E1 32213.642,E2 32213.642} C_VEL
LIN {X 0,Y 704.342,Z 393.482,A -85,B 0,C 180,E1 32210.769,E2 32210.769} C_VEL
LIN {X 0,Y 704.267,Z 393.498,A -85,B 0,C 180,E1 32207.953,E2 32207.953} C_VEL
LIN {X 0,Y 704.271,Z 393.49,A -85,B 0,C 180,E1 32205.446,E2 32205.446} C_VEL
LIN {X 0,Y 704.345,Z 393.495,A -85,B 0,C 180,E1 32202.526,E2 32202.526} C_VEL
LIN {X 0,Y 704.274,Z 393.483,A -85,B 0,C 180,E1 32199.645,E2 32199.645} C_VEL
LIN {X 0,Y 704.298,Z 393.493,A -85,B 0,C 180,E1 32197.911,E2 32197.911} C_VEL
LIN {X 0,Y 703.269,Z 393.623,A -85,B 0,C 180,E1 32197.284,E2 32197.284} C_VEL
LIN {X 0,Y 696.854,Z 394.427,A -85,B 0,C 180,E1 32195.528,E2 32195.528} C_VEL
LIN {X 0,Y 696.354,Z 394.483,A -85,B 0,C 180,E1 32195.072,E2 32195.072} C_VEL
LIN {X 0,Y 696.395,Z 394.481,A -85,B 0,C 180,E1 32191.995,E2 32191.995} C_VEL
LIN {X 0,Y 696.35,Z 394.471,A -85,B 0,C 180,E1 32189.154,E2 32189.154} C_VEL
LIN {X 0,Y 696.399,Z 394.472,A -85,B 0,C 180,E1 32186.244,E2 32186.244} C_VEL
LIN {X 0,Y 696.364,Z 394.485,A -85,B 0,C 180,E1 32183.321,E2 32183.321} C_VEL
LIN {X 0,Y 696.401,Z 394.479,A -85,B 0,C 180,E1 32180.395,E2 32180.395} C_VEL
LIN {X 0,Y 696.38,Z 394.482,A -85,B 0,C 180,E1 32177.311,E2 32177.311} C_VEL
LIN {X 0,Y 696.41,Z 394.595,A -85,B 0,C 180,E1 32175.836,E2 32175.836} C_VEL
LIN {X 0,Y 697.984,Z 398.359,A -85,B 0,C 180,E1 32175.431,E2 32175.431} C_VEL
LIN {X 0,Y 712.291,Z 419.94,A -85,B 0,C 180,E1 32173.975,E2 32173.975} C_VEL
LIN {X 0,Y 710.487,Z 625.213,A -85,B 0,C 180,E1 32171.347,E2 32171.347} C_VEL
LIN {X 0,Y 708.654,Z 849.902,A -85,B 0,C 180,E1 32168.563,E2 32168.563} C_VEL
LIN {X 0,Y 708.227,Z 883.584,A -85,B 0,C 180,E1 32168.107,E2 32168.107} C_VEL
LIN {X 0,Y 707.582,Z 910.326,A -85,B 0,C 180,E1 32167.583,E2 32167.583} C_VEL
LIN {X 0,Y 706.902,Z 935.438,A -85,B 0,C 180,E1 32166.942,E2 32166.942} C_VEL
LIN {X 0,Y 706.007,Z 963.024,A -85,B 0,C 180,E1 32166.058,E2 32166.058} C_VEL
LIN {X 0,Y 705.095,Z 986.74,A -85,B 0,C 180,E1 32165.145,E2 32165.145} C_VEL
LIN {X 0,Y 704.273,Z 1006.818,A -85,B 0,C 180,E1 32164.257,E2 32164.257} C_VEL
LIN {X 0,Y 703.421,Z 1026.605,A -85,B 0,C 180,E1 32163.27,E2 32163.27} C_VEL
LIN {X 0,Y 702.397,Z 1049.99,A -85,B 0,C 180,E1 32161.958,E2 32161.958} C_VEL
LIN {X 0,Y 701.386,Z 1072.697,A -85,B 0,C 180,E1 32160.492,E2 32160.492} C_VEL
LIN {X 0,Y 700.546,Z 1091.206,A -85,B 0,C 180,E1 32159.161,E2 32159.161} C_VEL
LIN {X 0,Y 699.716,Z 1110.481,A -85,B 0,C 180,E1 32157.628,E2 32157.628} C_VEL
LIN {X 0,Y 698.899,Z 1130.28,A -85,B 0,C 180,E1 32155.856,E2 32155.856} C_VEL
LIN {X 0,Y 698.264,Z 1146.311,A -85,B 0,C 180,E1 32154.26,E2 32154.26} C_VEL
LIN {X 0,Y 697.664,Z 1162.376,A -85,B 0,C 180,E1 32152.493,E2 32152.493} C_VEL
LIN {X 0,Y 697.115,Z 1179.227,A -85,B 0,C 180,E1 32150.393,E2 32150.393} C_VEL
LIN {X 0,Y 696.784,Z 1191.574,A -85,B 0,C 180,E1 32148.658,E2 32148.658} C_VEL
LIN {X 0,Y 696.499,Z 1203.069,A -85,B 0,C 180,E1 32146.852,E2 32146.852} C_VEL
LIN {X 0,Y 696.269,Z 1215.41,A -85,B 0,C 180,E1 32144.635,E2 32144.635} C_VEL
LIN {X 0,Y 696.097,Z 1225.262,A -85,B 0,C 180,E1 32142.522,E2 32142.522} C_VEL
LIN {X 0,Y 695.997,Z 1232.287,A -85,B 0,C 180,E1 32140.759,E2 32140.759} C_VEL
LIN {X 0,Y 695.917,Z 1237.925,A -85,B 0,C 180,E1 32139.089,E2 32139.089} C_VEL
LIN {X 0,Y 695.931,Z 1243.273,A -85,B 0,C 180,E1 32137.176,E2 32137.176} C_VEL
LIN {X 0,Y 695.918,Z 1247.856,A -85,B 0,C 180,E1 32134.941,E2 32134.941} C_VEL
LIN {X 0,Y 695.913,Z 1250.575,A -85,B 0,C 180,E1 32132.796,E2 32132.796} C_VEL
LIN {X 0,Y 695.876,Z 1251.726,A -85,B 0,C 180,E1 32130.984,E2 32130.984} C_VEL
LIN {X 0,Y 695.864,Z 1251.838,A -85,B 0,C 180,E1 32129.338,E2 32129.338} C_VEL
LIN {X 0,Y 695.904,Z 1250.98,A -85,B 0,C 180,E1 32127.608,E2 32127.608} C_VEL
LIN {X 0,Y 695.916,Z 1248.866,A -85,B 0,C 180,E1 32125.629,E2 32125.629} C_VEL
LIN {X 0,Y 695.925,Z 1244.821,A -85,B 0,C 180,E1 32123.396,E2 32123.396} C_VEL
LIN {X 0,Y 695.946,Z 1239.203,A -85,B 0,C 180,E1 32121.237,E2 32121.237} C_VEL
LIN {X 0,Y 695.995,Z 1233.201,A -85,B 0,C 180,E1 32119.4,E2 32119.4} C_VEL
LIN {X 0,Y 696.071,Z 1226.321,A -85,B 0,C 180,E1 32117.637,E2 32117.637} C_VEL
LIN {X 0,Y 696.186,Z 1218.27,A -85,B 0,C 180,E1 32115.865,E2 32115.865} C_VEL
LIN {X 0,Y 696.372,Z 1208.966,A -85,B 0,C 180,E1 32114.08,E2 32114.08} C_VEL
LIN {X 0,Y 696.662,Z 1195.597,A -85,B 0,C 180,E1 32111.85,E2 32111.85} C_VEL
LIN {X 0,Y 697.023,Z 1182.409,A -85,B 0,C 180,E1 32109.947,E2 32109.947} C_VEL
LIN {X 0,Y 697.435,Z 1169.55,A -85,B 0,C 180,E1 32108.283,E2 32108.283} C_VEL
LIN {X 0,Y 698.024,Z 1152.971,A -85,B 0,C 180,E1 32106.351,E2 32106.351} C_VEL
LIN {X 0,Y 698.711,Z 1134.745,A -85,B 0,C 180,E1 32104.483,E2 32104.483} C_VEL
LIN {X 0,Y 699.376,Z 1118.234,A -85,B 0,C 180,E1 32102.956,E2 32102.956} C_VEL
LIN {X 0,Y 700.282,Z 1097.643,A -85,B 0,C 180,E1 32101.235,E2 32101.235} C_VEL
LIN {X 0,Y 701.208,Z 1076.487,A -85,B 0,C 180,E1 32099.68,E2 32099.68} C_VEL
LIN {X 0,Y 702.058,Z 1057.717,A -85,B 0,C 180,E1 32098.437,E2 32098.437} C_VEL
LIN {X 0,Y 702.983,Z 1037.04,A -85,B 0,C 180,E1 32097.205,E2 32097.205} C_VEL
LIN {X 0,Y 704.057,Z 1011.533,A -85,B 0,C 180,E1 32095.875,E2 32095.875} C_VEL
LIN {X 0,Y 704.954,Z 989.79,A -85,B 0,C 180,E1 32094.893,E2 32094.893} C_VEL
LIN {X 0,Y 705.728,Z 969.39,A -85,B 0,C 180,E1 32094.084,E2 32094.084} C_VEL
LIN {X 0,Y 706.486,Z 947.193,A -85,B 0,C 180,E1 32093.324,E2 32093.324} C_VEL
LIN {X 0,Y 707.315,Z 921.427,A -85,B 0,C 180,E1 32092.59,E2 32092.59} C_VEL
LIN {X 0,Y 707.99,Z 894.214,A -85,B 0,C 180,E1 32091.994,E2 32091.994} C_VEL
LIN {X 0,Y 708.444,Z 869.295,A -85,B 0,C 180,E1 32091.59,E2 32091.59} C_VEL
LIN {X 0,Y 710.337,Z 642.37,A -85,B 0,C 180,E1 32088.779,E2 32088.779} C_VEL
LIN {X 0,Y 712.161,Z 435.225,A -85,B 0,C 180,E1 32086.134,E2 32086.134} C_VEL
LIN {X 0,Y 712.142,Z 419.653,A -85,B 0,C 180,E1 32085.919,E2 32085.919} C_VEL
LIN {X 0,Y 700.555,Z 402.372,A -85,B 0,C 180,E1 32084.75,E2 32084.75} C_VEL
LIN {X 0,Y 697.649,Z 397.879,A -85,B 0,C 180,E1 32084.438,E2 32084.438} C_VEL
LIN {X 0,Y 696.384,Z 394.489,A -85,B 0,C 180,E1 32084.044,E2 32084.044} C_VEL
LIN {X 0,Y 696.387,Z 394.489,A -85,B 0,C 180,E1 32081.077,E2 32081.077} C_VEL
LIN {X 0,Y 696.395,Z 394.482,A -85,B 0,C 180,E1 32078.109,E2 32078.109} C_VEL
LIN {X 0,Y 696.396,Z 394.472,A -85,B 0,C 180,E1 32075.052,E2 32075.052} C_VEL
LIN {X 0,Y 696.396,Z 394.479,A -85,B 0,C 180,E1 32071.943,E2 32071.943} C_VEL
LIN {X 0,Y 696.401,Z 394.481,A -85,B 0,C 180,E1 32068.844,E2 32068.844} C_VEL
LIN {X 0,Y 696.396,Z 394.465,A -85,B 0,C 180,E1 32065.789,E2 32065.789} C_VEL
LIN {X 0,Y 696.405,Z 394.488,A -85,B 0,C 180,E1 32062.72,E2 32062.72} C_VEL
LIN {X 0,Y 696.395,Z 394.468,A -85,B 0,C 180,E1 32059.545,E2 32059.545} C_VEL
LIN {X 0,Y 696.4,Z 394.48,A -85,B 0,C 180,E1 32056.431,E2 32056.431} C_VEL
LIN {X 0,Y 696.391,Z 394.473,A -85,B 0,C 180,E1 32053.281,E2 32053.281} C_VEL
LIN {X 0,Y 696.398,Z 394.477,A -85,B 0,C 180,E1 32050.256,E2 32050.256} C_VEL
LIN {X 0,Y 696.392,Z 394.475,A -85,B 0,C 180,E1 32047.093,E2 32047.093} C_VEL
LIN {X 0,Y 696.394,Z 394.476,A -85,B 0,C 180,E1 32044.034,E2 32044.034} C_VEL
LIN {X 0,Y 696.394,Z 394.475,A -85,B 0,C 180,E1 32040.905,E2 32040.905} C_VEL
LIN {X 0,Y 696.391,Z 394.476,A -85,B 0,C 180,E1 32037.861,E2 32037.861} C_VEL
LIN {X 0,Y 696.393,Z 394.476,A -85,B 0,C 180,E1 32034.728,E2 32034.728} C_VEL
LIN {X 0,Y 696.382,Z 394.478,A -85,B 0,C 180,E1 32031.745,E2 32031.745} C_VEL
LIN {X 0,Y 696.4,Z 394.477,A -85,B 0,C 180,E1 32028.656,E2 32028.656} C_VEL
LIN {X 0,Y 696.368,Z 394.479,A -85,B 0,C 180,E1 32025.702,E2 32025.702} C_VEL
LIN {X 0,Y 696.395,Z 394.483,A -85,B 0,C 180,E1 32022.796,E2 32022.796} C_VEL
LIN {X 0,Y 696.363,Z 394.469,A -85,B 0,C 180,E1 32019.842,E2 32019.842} C_VEL
LIN {X 0,Y 696.405,Z 394.486,A -85,B 0,C 180,E1 32016.923,E2 32016.923} C_VEL
LIN {X 0,Y 696.373,Z 394.475,A -85,B 0,C 180,E1 32013.821,E2 32013.821} C_VEL
LIN {X 0,Y 696.376,Z 394.48,A -85,B 0,C 180,E1 32010.967,E2 32010.967} C_VEL
LIN {X 0,Y 696.397,Z 394.48,A -85,B 0,C 180,E1 32007.902,E2 32007.902} C_VEL
LIN {X 0,Y 696.359,Z 394.481,A -85,B 0,C 180,E1 32005.046,E2 32005.046} C_VEL
LIN {X 0,Y 696.398,Z 394.472,A -85,B 0,C 180,E1 32002.158,E2 32002.158} C_VEL
LIN {X 0,Y 696.362,Z 394.489,A -85,B 0,C 180,E1 31999.177,E2 31999.177} C_VEL
LIN {X 0,Y 696.417,Z 394.605,A -85,B 0,C 180,E1 31998.115,E2 31998.115} C_VEL
LIN {X 0,Y 697.601,Z 397.807,A -85,B 0,C 180,E1 31997.76,E2 31997.76} C_VEL
LIN {X 0,Y 698.748,Z 400.196,A -85,B 0,C 180,E1 31997.474,E2 31997.474} C_VEL
LIN {X 0,Y 705.971,Z 415.441,A -85,B 0,C 180,E1 31995.713,E2 31995.713} C_VEL
LIN {X 0,Y 708.113,Z 420.435,A -85,B 0,C 180,E1 31995.174,E2 31995.174} C_VEL
LIN {X 0,Y 708.012,Z 428.141,A -85,B 0,C 180,E1 31994.66,E2 31994.66} C_VEL
LIN {X 0,Y 712.35,Z 445.49,A -85,B 0,C 180,E1 31994.077,E2 31994.077} C_VEL
LIN {X 0,Y 710.468,Z 657.167,A -85,B 0,C 180,E1 31991.367,E2 31991.367} C_VEL
LIN {X 0,Y 708.633,Z 882.598,A -85,B 0,C 180,E1 31988.575,E2 31988.575} C_VEL
LIN {X 0,Y 708.197,Z 914.752,A -85,B 0,C 180,E1 31988.132,E2 31988.132} C_VEL
LIN {X 0,Y 707.561,Z 941.01,A -85,B 0,C 180,E1 31987.612,E2 31987.612} C_VEL
LIN {X 0,Y 706.875,Z 966.295,A -85,B 0,C 180,E1 31986.962,E2 31986.962} C_VEL
LIN {X 0,Y 705.974,Z 993.817,A -85,B 0,C 180,E1 31986.074,E2 31986.074} C_VEL
LIN {X 0,Y 705.114,Z 1016.312,A -85,B 0,C 180,E1 31985.208,E2 31985.208} C_VEL
LIN {X 0,Y 704.281,Z 1036.648,A -85,B 0,C 180,E1 31984.31,E2 31984.31} C_VEL
LIN {X 0,Y 703.391,Z 1057.266,A -85,B 0,C 180,E1 31983.281,E2 31983.281} C_VEL
LIN {X 0,Y 702.367,Z 1080.805,A -85,B 0,C 180,E1 31981.954,E2 31981.954} C_VEL
LIN {X 0,Y 701.365,Z 1103.208,A -85,B 0,C 180,E1 31980.501,E2 31980.501} C_VEL
LIN {X 0,Y 700.555,Z 1121.012,A -85,B 0,C 180,E1 31979.22,E2 31979.22} C_VEL
LIN {X 0,Y 699.746,Z 1139.894,A -85,B 0,C 180,E1 31977.72,E2 31977.72} C_VEL
LIN {X 0,Y 698.879,Z 1160.783,A -85,B 0,C 180,E1 31975.853,E2 31975.853} C_VEL
LIN {X 0,Y 698.248,Z 1176.66,A -85,B 0,C 180,E1 31974.269,E2 31974.269} C_VEL
LIN {X 0,Y 697.634,Z 1193.468,A -85,B 0,C 180,E1 31972.413,E2 31972.413} C_VEL
LIN {X 0,Y 697.105,Z 1209.498,A -85,B 0,C 180,E1 31970.401,E2 31970.401} C_VEL
LIN {X 0,Y 696.779,Z 1221.821,A -85,B 0,C 180,E1 31968.666,E2 31968.666} C_VEL
LIN {X 0,Y 696.495,Z 1233.293,A -85,B 0,C 180,E1 31966.86,E2 31966.86} C_VEL
LIN {X 0,Y 696.265,Z 1245.589,A -85,B 0,C 180,E1 31964.643,E2 31964.643} C_VEL
LIN {X 0,Y 696.106,Z 1255.063,A -85,B 0,C 180,E1 31962.614,E2 31962.614} C_VEL
LIN {X 0,Y 695.995,Z 1262.119,A -85,B 0,C 180,E1 31960.851,E2 31960.851} C_VEL
LIN {X 0,Y 695.916,Z 1267.784,A -85,B 0,C 180,E1 31959.18,E2 31959.18} C_VEL
LIN {X 0,Y 695.919,Z 1272.958,A -85,B 0,C 180,E1 31957.35,E2 31957.35} C_VEL
LIN {X 0,Y 695.914,Z 1277.628,A -85,B 0,C 180,E1 31955.114,E2 31955.114} C_VEL
LIN {X 0,Y 695.91,Z 1280.47,A -85,B 0,C 180,E1 31952.969,E2 31952.969} C_VEL
LIN {X 0,Y 695.878,Z 1281.714,A -85,B 0,C 180,E1 31951.074,E2 31951.074} C_VEL
LIN {X 0,Y 695.863,Z 1281.828,A -85,B 0,C 180,E1 31949.345,E2 31949.345} C_VEL
LIN {X 0,Y 695.907,Z 1280.949,A -85,B 0,C 180,E1 31947.616,E2 31947.616} C_VEL
LIN {X 0,Y 695.917,Z 1278.854,A -85,B 0,C 180,E1 31945.667,E2 31945.667} C_VEL
LIN {X 0,Y 695.925,Z 1274.743,A -85,B 0,C 180,E1 31943.404,E2 31943.404} C_VEL
LIN {X 0,Y 695.941,Z 1269.088,A -85,B 0,C 180,E1 31941.244,E2 31941.244} C_VEL
LIN {X 0,Y 695.996,Z 1263.064,A -85,B 0,C 180,E1 31939.408,E2 31939.408} C_VEL
LIN {X 0,Y 696.062,Z 1256.525,A -85,B 0,C 180,E1 31937.73,E2 31937.73} C_VEL
LIN {X 0,Y 696.174,Z 1248.5,A -85,B 0,C 180,E1 31935.957,E2 31935.957} C_VEL
LIN {X 0,Y 696.368,Z 1239.231,A -85,B 0,C 180,E1 31934.173,E2 31934.173} C_VEL
LIN {X 0,Y 696.639,Z 1226.5,A -85,B 0,C 180,E1 31932.031,E2 31932.031} C_VEL
LIN {X 0,Y 697.014,Z 1212.781,A -85,B 0,C 180,E1 31930.042,E2 31930.042} C_VEL
LIN {X 0,Y 697.451,Z 1199.158,A -85,B 0,C 180,E1 31928.28,E2 31928.28} C_VEL
LIN {X 0,Y 698.039,Z 1182.65,A -85,B 0,C 180,E1 31926.36,E2 31926.36} C_VEL
LIN {X 0,Y 698.729,Z 1164.369,A -85,B 0,C 180,E1 31924.492,E2 31924.492} C_VEL
LIN {X 0,Y 699.397,Z 1147.754,A -85,B 0,C 180,E1 31922.958,E2 31922.958} C_VEL
LIN {X 0,Y 700.3,Z 1127.163,A -85,B 0,C 180,E1 31921.244,E2 31921.244} C_VEL
LIN {X 0,Y 701.2,Z 1106.638,A -85,B 0,C 180,E1 31919.736,E2 31919.736} C_VEL
LIN {X 0,Y 702.048,Z 1087.89,A -85,B 0,C 180,E1 31918.493,E2 31918.493} C_VEL
LIN {X 0,Y 702.951,Z 1067.694,A -85,B 0,C 180,E1 31917.288,E2 31917.288} C_VEL
LIN {X 0,Y 704.047,Z 1041.799,A -85,B 0,C 180,E1 31915.932,E2 31915.932} C_VEL
LIN {X 0,Y 704.945,Z 1019.989,A -85,B 0,C 180,E1 31914.946,E2 31914.946} C_VEL
LIN {X 0,Y 705.769,Z 998.481,A -85,B 0,C 180,E1 31914.096,E2 31914.096} C_VEL
LIN {X 0,Y 706.576,Z 974.666,A -85,B 0,C 180,E1 31913.288,E2 31913.288} C_VEL
LIN {X 0,Y 707.407,Z 947.885,A -85,B 0,C 180,E1 31912.549,E2 31912.549} C_VEL
LIN {X 0,Y 708.022,Z 922.429,A -85,B 0,C 180,E1 31912.005,E2 31912.005} C_VEL
LIN {X 0,Y 708.49,Z 896.642,A -85,B 0,C 180,E1 31911.599,E2 31911.599} C_VEL
LIN {X 0,Y 710.366,Z 669.057,A -85,B 0,C 180,E1 31908.782,E2 31908.782} C_VEL
LIN {X 0,Y 712.214,Z 459.951,A -85,B 0,C 180,E1 31906.111,E2 31906.111} C_VEL
LIN {X 0,Y 712.194,Z 444.186,A -85,B 0,C 180,E1 31905.893,E2 31905.893} C_VEL
LIN {X 0,Y 707.886,Z 427.36,A -85,B 0,C 180,E1 31905.306,E2 31905.306} C_VEL
LIN {X 0,Y 708.07,Z 420.145,A -85,B 0,C 180,E1 31904.802,E2 31904.802} C_VEL
LIN {X 0,Y 701.754,Z 406.449,A -85,B 0,C 180,E1 31903.263,E2 31903.263} C_VEL
LIN {X 0,Y 698.006,Z 398.382,A -85,B 0,C 180,E1 31902.32,E2 31902.32} C_VEL
LIN {X 0,Y 696.531,Z 395.213,A -85,B 0,C 180,E1 31901.942,E2 31901.942} C_VEL
LIN {X 0,Y 696.397,Z 394.479,A -85,B 0,C 180,E1 31901.835,E2 31901.835} C_VEL
LIN {X 0,Y 696.341,Z 394.49,A -85,B 0,C 180,E1 31899.039,E2 31899.039} C_VEL
LIN {X 0,Y 696.401,Z 394.48,A -85,B 0,C 180,E1 31896.165,E2 31896.165} C_VEL
LIN {X 0,Y 696.344,Z 394.483,A -85,B 0,C 180,E1 31893.266,E2 31893.266} C_VEL
LIN {X 0,Y 696.333,Z 394.482,A -85,B 0,C 180,E1 31890.648,E2 31890.648} C_VEL
LIN {X 0,Y 696.405,Z 394.484,A -85,B 0,C 180,E1 31887.723,E2 31887.723} C_VEL
LIN {X 0,Y 696.32,Z 394.48,A -85,B 0,C 180,E1 31884.85,E2 31884.85} C_VEL
LIN {X 0,Y 696.326,Z 394.488,A -85,B 0,C 180,E1 31882.366,E2 31882.366} C_VEL
LIN {X 0,Y 696.388,Z 394.475,A -85,B 0,C 180,E1 31879.401,E2 31879.401} C_VEL
LIN {X 0,Y 696.311,Z 394.487,A -85,B 0,C 180,E1 31876.69,E2 31876.69} C_VEL
LIN {X 0,Y 696.302,Z 394.477,A -85,B 0,C 180,E1 31874.3,E2 31874.3} C_VEL
LIN {X 0,Y 696.348,Z 394.49,A -85,B 0,C 180,E1 31871.681,E2 31871.681} C_VEL
LIN {X 0,Y 696.308,Z 394.481,A -85,B 0,C 180,E1 31868.672,E2 31868.672} C_VEL
LIN {X 0,Y 696.293,Z 394.491,A -85,B 0,C 180,E1 31866.266,E2 31866.266} C_VEL
LIN {X 0,Y 696.31,Z 394.483,A -85,B 0,C 180,E1 31863.787,E2 31863.787} C_VEL
LIN {X 0,Y 696.353,Z 394.489,A -85,B 0,C 180,E1 31860.74,E2 31860.74} C_VEL
LIN {X 0,Y 696.306,Z 394.481,A -85,B 0,C 180,E1 31858.107,E2 31858.107} C_VEL
LIN {X 0,Y 696.321,Z 394.48,A -85,B 0,C 180,E1 31855.635,E2 31855.635} C_VEL
LIN {X 0,Y 696.385,Z 394.477,A -85,B 0,C 180,E1 31852.658,E2 31852.658} C_VEL
LIN {X 0,Y 696.32,Z 394.479,A -85,B 0,C 180,E1 31849.91,E2 31849.91} C_VEL
LIN {X 0,Y 696.336,Z 394.489,A -85,B 0,C 180,E1 31847.393,E2 31847.393} C_VEL
LIN {X 0,Y 696.394,Z 394.475,A -85,B 0,C 180,E1 31844.425,E2 31844.425} C_VEL
LIN {X 0,Y 696.334,Z 394.486,A -85,B 0,C 180,E1 31841.628,E2 31841.628} C_VEL
LIN {X 0,Y 696.379,Z 394.472,A -85,B 0,C 180,E1 31838.875,E2 31838.875} C_VEL
LIN {X 0,Y 696.359,Z 394.48,A -85,B 0,C 180,E1 31835.844,E2 31835.844} C_VEL
LIN {X 0,Y 696.354,Z 394.483,A -85,B 0,C 180,E1 31835.072,E2 31835.072} C_VEL
LIN {X 0,Y 695.402,Z 394.597,A -85,B 0,C 180,E1 31834.438,E2 31834.438} C_VEL
LIN {X 0,Y 688.99,Z 395.41,A -85,B 0,C 180,E1 31832.662,E2 31832.662} C_VEL
LIN {X 0,Y 688.467,Z 395.472,A -85,B 0,C 180,E1 31832.201,E2 31832.201} C_VEL
LIN {X 0,Y 688.411,Z 395.457,A -85,B 0,C 180,E1 31829.287,E2 31829.287} C_VEL
LIN {X 0,Y 688.464,Z 395.463,A -85,B 0,C 180,E1 31826.403,E2 31826.403} C_VEL
LIN {X 0,Y 688.427,Z 395.474,A -85,B 0,C 180,E1 31823.348,E2 31823.348} C_VEL
LIN {X 0,Y 688.462,Z 395.467,A -85,B 0,C 180,E1 31820.388,E2 31820.388} C_VEL
LIN {X 0,Y 688.439,Z 395.472,A -85,B 0,C 180,E1 31817.291,E2 31817.291} C_VEL
LIN {X 0,Y 688.477,Z 395.647,A -85,B 0,C 180,E1 31816.436,E2 31816.436} C_VEL
LIN {X 0,Y 689.519,Z 398.57,A -85,B 0,C 180,E1 31816.148,E2 31816.148} C_VEL
LIN {X 0,Y 694.922,Z 406.34,A -85,B 0,C 180,E1 31815.573,E2 31815.573} C_VEL
LIN {X 0,Y 706.346,Z 423.321,A -85,B 0,C 180,E1 31814.396,E2 31814.396} C_VEL
LIN {X 0,Y 705.212,Z 550.164,A -85,B 0,C 180,E1 31812.738,E2 31812.738} C_VEL
LIN {X 0,Y 703.134,Z 767.426,A -85,B 0,C 180,E1 31809.992,E2 31809.992} C_VEL
LIN {X 0,Y 702.033,Z 877.114,A -85,B 0,C 180,E1 31808.615,E2 31808.615} C_VEL
LIN {X 0,Y 701.369,Z 905.145,A -85,B 0,C 180,E1 31808.101,E2 31808.101} C_VEL
LIN {X 0,Y 700.573,Z 930.656,A -85,B 0,C 180,E1 31807.474,E2 31807.474} C_VEL
LIN {X 0,Y 699.712,Z 953.683,A -85,B 0,C 180,E1 31806.773,E2 31806.773} C_VEL
LIN {X 0,Y 698.71,Z 979.972,A -85,B 0,C 180,E1 31805.817,E2 31805.817} C_VEL
LIN {X 0,Y 697.609,Z 1003.936,A -85,B 0,C 180,E1 31804.775,E2 31804.775} C_VEL
LIN {X 0,Y 696.652,Z 1023.76,A -85,B 0,C 180,E1 31803.795,E2 31803.795} C_VEL
LIN {X 0,Y 695.674,Z 1043.403,A -85,B 0,C 180,E1 31802.706,E2 31802.706} C_VEL
LIN {X 0,Y 694.592,Z 1064.659,A -85,B 0,C 180,E1 31801.389,E2 31801.389} C_VEL
LIN {X 0,Y 693.406,Z 1087.742,A -85,B 0,C 180,E1 31799.763,E2 31799.763} C_VEL
LIN {X 0,Y 692.528,Z 1105.59,A -85,B 0,C 180,E1 31798.354,E2 31798.354} C_VEL
LIN {X 0,Y 691.674,Z 1123.426,A -85,B 0,C 180,E1 31796.804,E2 31796.804} C_VEL
LIN {X 0,Y 690.719,Z 1143.759,A -85,B 0,C 180,E1 31794.817,E2 31794.817} C_VEL
LIN {X 0,Y 690.068,Z 1159.282,A -85,B 0,C 180,E1 31793.115,E2 31793.115} C_VEL
LIN {X 0,Y 689.475,Z 1175.298,A -85,B 0,C 180,E1 31791.163,E2 31791.163} C_VEL
LIN {X 0,Y 688.967,Z 1190.416,A -85,B 0,C 180,E1 31789.054,E2 31789.054} C_VEL
LIN {X 0,Y 688.615,Z 1202.03,A -85,B 0,C 180,E1 31787.225,E2 31787.225} C_VEL
LIN {X 0,Y 688.351,Z 1212.804,A -85,B 0,C 180,E1 31785.307,E2 31785.307} C_VEL
LIN {X 0,Y 688.146,Z 1223.836,A -85,B 0,C 180,E1 31783.011,E2 31783.011} C_VEL
LIN {X 0,Y 688.024,Z 1231.678,A -85,B 0,C 180,E1 31781.055,E2 31781.055} C_VEL
LIN {X 0,Y 687.926,Z 1237.671,A -85,B 0,C 180,E1 31779.28,E2 31779.28} C_VEL
LIN {X 0,Y 687.916,Z 1242.863,A -85,B 0,C 180,E1 31777.428,E2 31777.428} C_VEL
LIN {X 0,Y 687.914,Z 1247.413,A -85,B 0,C 180,E1 31775.25,E2 31775.25} C_VEL
LIN {X 0,Y 687.909,Z 1250.387,A -85,B 0,C 180,E1 31773.06,E2 31773.06} C_VEL
LIN {X 0,Y 687.884,Z 1251.704,A -85,B 0,C 180,E1 31771.079,E2 31771.079} C_VEL
LIN {X 0,Y 687.864,Z 1251.838,A -85,B 0,C 180,E1 31769.33,E2 31769.33} C_VEL
LIN {X 0,Y 687.903,Z 1250.98,A -85,B 0,C 180,E1 31767.58,E2 31767.58} C_VEL
LIN {X 0,Y 687.914,Z 1248.865,A -85,B 0,C 180,E1 31765.578,E2 31765.578} C_VEL
LIN {X 0,Y 687.925,Z 1244.82,A -85,B 0,C 180,E1 31763.319,E2 31763.319} C_VEL
LIN {X 0,Y 687.941,Z 1239.202,A -85,B 0,C 180,E1 31761.134,E2 31761.134} C_VEL
LIN {X 0,Y 688.002,Z 1233.109,A -85,B 0,C 180,E1 31759.251,E2 31759.251} C_VEL
LIN {X 0,Y 688.108,Z 1226.325,A -85,B 0,C 180,E1 31757.493,E2 31757.493} C_VEL
LIN {X 0,Y 688.248,Z 1218.268,A -85,B 0,C 180,E1 31755.698,E2 31755.698} C_VEL
LIN {X 0,Y 688.447,Z 1208.499,A -85,B 0,C 180,E1 31753.805,E2 31753.805} C_VEL
LIN {X 0,Y 688.818,Z 1195.018,A -85,B 0,C 180,E1 31751.549,E2 31751.549} C_VEL
LIN {X 0,Y 689.196,Z 1182.406,A -85,B 0,C 180,E1 31749.709,E2 31749.709} C_VEL
LIN {X 0,Y 689.7,Z 1168.884,A -85,B 0,C 180,E1 31747.943,E2 31747.943} C_VEL
LIN {X 0,Y 690.407,Z 1151.32,A -85,B 0,C 180,E1 31745.892,E2 31745.892} C_VEL
LIN {X 0,Y 691.205,Z 1133.447,A -85,B 0,C 180,E1 31744.057,E2 31744.057} C_VEL
LIN {X 0,Y 691.981,Z 1116.195,A -85,B 0,C 180,E1 31742.456,E2 31742.456} C_VEL
LIN {X 0,Y 693.102,Z 1093.901,A -85,B 0,C 180,E1 31740.616,E2 31740.616} C_VEL
LIN {X 0,Y 694.062,Z 1075.155,A -85,B 0,C 180,E1 31739.239,E2 31739.239} C_VEL
LIN {X 0,Y 695.016,Z 1056.246,A -85,B 0,C 180,E1 31737.982,E2 31737.982} C_VEL
LIN {X 0,Y 696.24,Z 1032.063,A -85,B 0,C 180,E1 31736.553,E2 31736.553} C_VEL
LIN {X 0,Y 697.344,Z 1009.329,A -85,B 0,C 180,E1 31735.39,E2 31735.39} C_VEL
LIN {X 0,Y 698.25,Z 989.667,A -85,B 0,C 180,E1 31734.5,E2 31734.5} C_VEL
LIN {X 0,Y 699.118,Z 969.377,A -85,B 0,C 180,E1 31733.691,E2 31733.691} C_VEL
LIN {X 0,Y 699.961,Z 947.171,A -85,B 0,C 180,E1 31732.925,E2 31732.925} C_VEL
LIN {X 0,Y 700.895,Z 921.441,A -85,B 0,C 180,E1 31732.188,E2 31732.188} C_VEL
LIN {X 0,Y 701.648,Z 894.182,A -85,B 0,C 180,E1 31731.588,E2 31731.588} C_VEL
LIN {X 0,Y 702.156,Z 869.439,A -85,B 0,C 180,E1 31731.186,E2 31731.186} C_VEL
LIN {X 0,Y 704.288,Z 644.481,A -85,B 0,C 180,E1 31728.375,E2 31728.375} C_VEL
LIN {X 0,Y 706.359,Z 437.211,A -85,B 0,C 180,E1 31725.708,E2 31725.708} C_VEL
LIN {X 0,Y 706.356,Z 423.332,A -85,B 0,C 180,E1 31725.515,E2 31725.515} C_VEL
LIN {X 0,Y 692.937,Z 403.355,A -85,B 0,C 180,E1 31724.126,E2 31724.126} C_VEL
LIN {X 0,Y 689.051,Z 397.667,A -85,B 0,C 180,E1 31723.688,E2 31723.688} C_VEL
LIN {X 0,Y 688.462,Z 395.477,A -85,B 0,C 180,E1 31723.431,E2 31723.431} C_VEL
LIN {X 0,Y 688.463,Z 395.471,A -85,B 0,C 180,E1 31720.263,E2 31720.263} C_VEL
LIN {X 0,Y 688.458,Z 395.474,A -85,B 0,C 180,E1 31717.121,E2 31717.121} C_VEL
LIN {X 0,Y 688.455,Z 395.457,A -85,B 0,C 180,E1 31713.998,E2 31713.998} C_VEL
LIN {X 0,Y 688.461,Z 395.459,A -85,B 0,C 180,E1 31710.94,E2 31710.94} C_VEL
LIN {X 0,Y 688.457,Z 395.468,A -85,B 0,C 180,E1 31707.789,E2 31707.789} C_VEL
LIN {X 0,Y 688.458,Z 395.461,A -85,B 0,C 180,E1 31704.726,E2 31704.726} C_VEL
LIN {X 0,Y 688.459,Z 395.462,A -85,B 0,C 180,E1 31701.64,E2 31701.64} C_VEL
LIN {X 0,Y 688.46,Z 395.47,A -85,B 0,C 180,E1 31698.546,E2 31698.546} C_VEL
LIN {X 0,Y 688.456,Z 395.455,A -85,B 0,C 180,E1 31695.414,E2 31695.414} C_VEL
LIN {X 0,Y 688.461,Z 395.474,A -85,B 0,C 180,E1 31692.327,E2 31692.327} C_VEL
LIN {X 0,Y 688.453,Z 395.45,A -85,B 0,C 180,E1 31689.193,E2 31689.193} C_VEL
LIN {X 0,Y 688.461,Z 395.476,A -85,B 0,C 180,E1 31686.086,E2 31686.086} C_VEL
LIN {X 0,Y 688.446,Z 395.448,A -85,B 0,C 180,E1 31682.914,E2 31682.914} C_VEL
LIN {X 0,Y 688.468,Z 395.476,A -85,B 0,C 180,E1 31679.834,E2 31679.834} C_VEL
LIN {X 0,Y 688.443,Z 395.447,A -85,B 0,C 180,E1 31676.669,E2 31676.669} C_VEL
LIN {X 0,Y 688.458,Z 395.476,A -85,B 0,C 180,E1 31673.663,E2 31673.663} C_VEL
LIN {X 0,Y 688.451,Z 395.449,A -85,B 0,C 180,E1 31670.554,E2 31670.554} C_VEL
LIN {X 0,Y 688.45,Z 395.477,A -85,B 0,C 180,E1 31667.502,E2 31667.502} C_VEL
LIN {X 0,Y 688.449,Z 395.458,A -85,B 0,C 180,E1 31664.327,E2 31664.327} C_VEL
LIN {X 0,Y 688.442,Z 395.476,A -85,B 0,C 180,E1 31661.366,E2 31661.366} C_VEL
LIN {X 0,Y 688.464,Z 395.466,A -85,B 0,C 180,E1 31658.263,E2 31658.263} C_VEL
LIN {X 0,Y 688.425,Z 395.467,A -85,B 0,C 180,E1 31655.364,E2 31655.364} C_VEL
LIN {X 0,Y 688.46,Z 395.471,A -85,B 0,C 180,E1 31652.369,E2 31652.369} C_VEL
LIN {X 0,Y 688.422,Z 395.464,A -85,B 0,C 180,E1 31649.446,E2 31649.446} C_VEL
LIN {X 0,Y 688.459,Z 395.459,A -85,B 0,C 180,E1 31646.503,E2 31646.503} C_VEL
LIN {X 0,Y 688.43,Z 395.47,A -85,B 0,C 180,E1 31643.437,E2 31643.437} C_VEL
LIN {X 0,Y 688.436,Z 395.479,A -85,B 0,C 180,E1 31640.597,E2 31640.597} C_VEL
LIN {X 0,Y 688.44,Z 395.62,A -85,B 0,C 180,E1 31638.773,E2 31638.773} C_VEL
LIN {X 0,Y 689.73,Z 398.924,A -85,B 0,C 180,E1 31638.398,E2 31638.398} C_VEL
LIN {X 0,Y 690.781,Z 400.937,A -85,B 0,C 180,E1 31638.142,E2 31638.142} C_VEL
LIN {X 0,Y 699.761,Z 419.936,A -85,B 0,C 180,E1 31635.903,E2 31635.903} C_VEL
LIN {X 0,Y 701.683,Z 424.559,A -85,B 0,C 180,E1 31635.402,E2 31635.402} C_VEL
LIN {X 0,Y 701.691,Z 428.114,A -85,B 0,C 180,E1 31635.173,E2 31635.173} C_VEL
LIN {X 0,Y 706.568,Z 447.731,A -85,B 0,C 180,E1 31634.502,E2 31634.502} C_VEL
LIN {X 0,Y 704.442,Z 658.771,A -85,B 0,C 180,E1 31631.779,E2 31631.779} C_VEL
LIN {X 0,Y 702.359,Z 884.075,A -85,B 0,C 180,E1 31628.965,E2 31628.965} C_VEL
LIN {X 0,Y 701.854,Z 915.906,A -85,B 0,C 180,E1 31628.518,E2 31628.518} C_VEL
LIN {X 0,Y 701.156,Z 941.563,A -85,B 0,C 180,E1 31628.002,E2 31628.002} C_VEL
LIN {X 0,Y 700.377,Z 966.874,A -85,B 0,C 180,E1 31627.345,E2 31627.345} C_VEL
LIN {X 0,Y 699.351,Z 994.392,A -85,B 0,C 180,E1 31626.448,E2 31626.448} C_VEL
LIN {X 0,Y 698.407,Z 1016.442,A -85,B 0,C 180,E1 31625.591,E2 31625.591} C_VEL
LIN {X 0,Y 697.477,Z 1036.652,A -85,B 0,C 180,E1 31624.692,E2 31624.692} C_VEL
LIN {X 0,Y 696.518,Z 1056.379,A -85,B 0,C 180,E1 31623.702,E2 31623.702} C_VEL
LIN {X 0,Y 695.398,Z 1078.888,A -85,B 0,C 180,E1 31622.432,E2 31622.432} C_VEL
LIN {X 0,Y 694.189,Z 1102.542,A -85,B 0,C 180,E1 31620.899,E2 31620.899} C_VEL
LIN {X 0,Y 693.241,Z 1121.013,A -85,B 0,C 180,E1 31619.559,E2 31619.559} C_VEL
LIN {X 0,Y 692.343,Z 1139.636,A -85,B 0,C 180,E1 31618.065,E2 31618.065} C_VEL
LIN {X 0,Y 691.321,Z 1160.557,A -85,B 0,C 180,E1 31616.179,E2 31616.179} C_VEL
LIN {X 0,Y 690.613,Z 1176.661,A -85,B 0,C 180,E1 31614.555,E2 31614.555} C_VEL
LIN {X 0,Y 689.9,Z 1193.464,A -85,B 0,C 180,E1 31612.679,E2 31612.679} C_VEL
LIN {X 0,Y 689.299,Z 1209.5,A -85,B 0,C 180,E1 31610.643,E2 31610.643} C_VEL
LIN {X 0,Y 688.912,Z 1222.016,A -85,B 0,C 180,E1 31608.858,E2 31608.858} C_VEL
LIN {X 0,Y 688.581,Z 1233.816,A -85,B 0,C 180,E1 31606.973,E2 31606.973} C_VEL
LIN {X 0,Y 688.299,Z 1246.411,A -85,B 0,C 180,E1 31604.644,E2 31604.644} C_VEL
LIN {X 0,Y 688.133,Z 1255.422,A -85,B 0,C 180,E1 31602.678,E2 31602.678} C_VEL
LIN {X 0,Y 688.008,Z 1262.425,A -85,B 0,C 180,E1 31600.894,E2 31600.894} C_VEL
LIN {X 0,Y 687.922,Z 1268.041,A -85,B 0,C 180,E1 31599.203,E2 31599.203} C_VEL
LIN {X 0,Y 687.922,Z 1273.162,A -85,B 0,C 180,E1 31597.352,E2 31597.352} C_VEL
LIN {X 0,Y 687.916,Z 1277.776,A -85,B 0,C 180,E1 31595.09,E2 31595.09} C_VEL
LIN {X 0,Y 687.912,Z 1280.538,A -85,B 0,C 180,E1 31592.92,E2 31592.92} C_VEL
LIN {X 0,Y 687.879,Z 1281.714,A -85,B 0,C 180,E1 31591.086,E2 31591.086} C_VEL
LIN {X 0,Y 687.863,Z 1281.828,A -85,B 0,C 180,E1 31589.338,E2 31589.338} C_VEL
LIN {X 0,Y 687.907,Z 1280.949,A -85,B 0,C 180,E1 31587.588,E2 31587.588} C_VEL
LIN {X 0,Y 687.916,Z 1278.892,A -85,B 0,C 180,E1 31585.643,E2 31585.643} C_VEL
LIN {X 0,Y 687.926,Z 1274.743,A -85,B 0,C 180,E1 31583.327,E2 31583.327} C_VEL
LIN {X 0,Y 687.938,Z 1269.089,A -85,B 0,C 180,E1 31581.142,E2 31581.142} C_VEL
LIN {X 0,Y 688.006,Z 1263.065,A -85,B 0,C 180,E1 31579.284,E2 31579.284} C_VEL
LIN {X 0,Y 688.111,Z 1256.169,A -85,B 0,C 180,E1 31577.5,E2 31577.5} C_VEL
LIN {X 0,Y 688.255,Z 1248.062,A -85,B 0,C 180,E1 31575.7,E2 31575.7} C_VEL
LIN {X 0,Y 688.459,Z 1237.836,A -85,B 0,C 180,E1 31573.727,E2 31573.727} C_VEL
LIN {X 0,Y 688.859,Z 1223.831,A -85,B 0,C 180,E1 31571.414,E2 31571.414} C_VEL
LIN {X 0,Y 689.237,Z 1211.144,A -85,B 0,C 180,E1 31569.582,E2 31569.582} C_VEL
LIN {X 0,Y 689.796,Z 1196.461,A -85,B 0,C 180,E1 31567.685,E2 31567.685} C_VEL
LIN {X 0,Y 690.542,Z 1178.267,A -85,B 0,C 180,E1 31565.614,E2 31565.614} C_VEL
LIN {X 0,Y 691.245,Z 1162.506,A -85,B 0,C 180,E1 31564.011,E2 31564.011} C_VEL
LIN {X 0,Y 692.117,Z 1143.767,A -85,B 0,C 180,E1 31562.284,E2 31562.284} C_VEL
LIN {X 0,Y 693.135,Z 1123.245,A -85,B 0,C 180,E1 31560.611,E2 31560.611} C_VEL
LIN {X 0,Y 694.084,Z 1104.652,A -85,B 0,C 180,E1 31559.249,E2 31559.249} C_VEL
LIN {X 0,Y 695.096,Z 1084.504,A -85,B 0,C 180,E1 31557.917,E2 31557.917} C_VEL
LIN {X 0,Y 696.378,Z 1059.211,A -85,B 0,C 180,E1 31556.447,E2 31556.447} C_VEL
LIN {X 0,Y 697.398,Z 1038.246,A -85,B 0,C 180,E1 31555.384,E2 31555.384} C_VEL
LIN {X 0,Y 698.289,Z 1018.875,A -85,B 0,C 180,E1 31554.511,E2 31554.511} C_VEL
LIN {X 0,Y 699.16,Z 998.48,A -85,B 0,C 180,E1 31553.703,E2 31553.703} C_VEL
LIN {X 0,Y 700.031,Z 975.403,A -85,B 0,C 180,E1 31552.914,E2 31552.914} C_VEL
LIN {X 0,Y 700.969,Z 948.873,A -85,B 0,C 180,E1 31552.171,E2 31552.171} C_VEL
LIN {X 0,Y 701.671,Z 923.052,A -85,B 0,C 180,E1 31551.612,E2 31551.612} C_VEL
LIN {X 0,Y 702.191,Z 897.824,A -85,B 0,C 180,E1 31551.208,E2 31551.208} C_VEL
LIN {X 0,Y 704.324,Z 670.866,A -85,B 0,C 180,E1 31548.374,E2 31548.374} C_VEL
LIN {X 0,Y 706.421,Z 461.695,A -85,B 0,C 180,E1 31545.681,E2 31545.681} C_VEL
LIN {X 0,Y 706.416,Z 446.394,A -85,B 0,C 180,E1 31545.468,E2 31545.468} C_VEL
LIN {X 0,Y 701.575,Z 427.36,A -85,B 0,C 180,E1 31544.794,E2 31544.794} C_VEL
LIN {X 0,Y 701.496,Z 423.84,A -85,B 0,C 180,E1 31544.53,E2 31544.53} C_VEL
LIN {X 0,Y 693.823,Z 407.397,A -85,B 0,C 180,E1 31542.636,E2 31542.636} C_VEL
LIN {X 0,Y 690.133,Z 399.479,A -85,B 0,C 180,E1 31541.684,E2 31541.684} C_VEL
LIN {X 0,Y 688.529,Z 396.17,A -85,B 0,C 180,E1 31541.278,E2 31541.278} C_VEL
LIN {X 0,Y 688.406,Z 395.461,A -85,B 0,C 180,E1 31541.187,E2 31541.187} C_VEL
LIN {X 0,Y 688.455,Z 395.466,A -85,B 0,C 180,E1 31538.328,E2 31538.328} C_VEL
LIN {X 0,Y 688.409,Z 395.475,A -85,B 0,C 180,E1 31535.297,E2 31535.297} C_VEL
LIN {X 0,Y 688.397,Z 395.473,A -85,B 0,C 180,E1 31532.706,E2 31532.706} C_VEL
LIN {X 0,Y 688.467,Z 395.457,A -85,B 0,C 180,E1 31529.729,E2 31529.729} C_VEL
LIN {X 0,Y 688.387,Z 395.475,A -85,B 0,C 180,E1 31526.855,E2 31526.855} C_VEL
LIN {X 0,Y 688.398,Z 395.466,A -85,B 0,C 180,E1 31524.271,E2 31524.271} C_VEL
LIN {X 0,Y 688.403,Z 395.464,A -85,B 0,C 180,E1 31521.113,E2 31521.113} C_VEL
LIN {X 0,Y 688.371,Z 395.476,A -85,B 0,C 180,E1 31518.549,E2 31518.549} C_VEL
LIN {X 0,Y 688.389,Z 395.475,A -85,B 0,C 180,E1 31516.02,E2 31516.02} C_VEL
LIN {X 0,Y 688.384,Z 395.48,A -85,B 0,C 180,E1 31512.84,E2 31512.84} C_VEL
LIN {X 0,Y 688.356,Z 395.473,A -85,B 0,C 180,E1 31510.292,E2 31510.292} C_VEL
LIN {X 0,Y 688.378,Z 395.469,A -85,B 0,C 180,E1 31507.764,E2 31507.764} C_VEL
LIN {X 0,Y 688.382,Z 395.471,A -85,B 0,C 180,E1 31504.666,E2 31504.666} C_VEL
LIN {X 0,Y 688.359,Z 395.469,A -85,B 0,C 180,E1 31502.164,E2 31502.164} C_VEL
LIN {X 0,Y 688.375,Z 395.479,A -85,B 0,C 180,E1 31499.75,E2 31499.75} C_VEL
LIN {X 0,Y 688.436,Z 395.459,A -85,B 0,C 180,E1 31496.753,E2 31496.753} C_VEL
LIN {X 0,Y 688.376,Z 395.478,A -85,B 0,C 180,E1 31493.997,E2 31493.997} C_VEL
LIN {X 0,Y 688.39,Z 395.468,A -85,B 0,C 180,E1 31491.506,E2 31491.506} C_VEL
LIN {X 0,Y 688.435,Z 395.474,A -85,B 0,C 180,E1 31488.438,E2 31488.438} C_VEL
LIN {X 0,Y 688.387,Z 395.465,A -85,B 0,C 180,E1 31485.704,E2 31485.704} C_VEL
LIN {X 0,Y 688.431,Z 395.472,A -85,B 0,C 180,E1 31483.026,E2 31483.026} C_VEL
LIN {X 0,Y 688.415,Z 395.456,A -85,B 0,C 180,E1 31479.954,E2 31479.954} C_VEL
LIN {X 0,Y 688.406,Z 395.475,A -85,B 0,C 180,E1 31477.249,E2 31477.249} C_VEL
LIN {X 0,Y 688.462,Z 395.457,A -85,B 0,C 180,E1 31474.262,E2 31474.262} C_VEL
LIN {X 0,Y 688.467,Z 395.472,A -85,B 0,C 180,E1 31472.201,E2 31472.201} C_VEL
LIN {X 0,Y 687.486,Z 395.59,A -85,B 0,C 180,E1 31471.56,E2 31471.56} C_VEL
LIN {X 0,Y 681.014,Z 396.379,A -85,B 0,C 180,E1 31469.764,E2 31469.764} C_VEL
LIN {X 0,Y 680.473,Z 396.445,A -85,B 0,C 180,E1 31469.296,E2 31469.296} C_VEL
LIN {X 0,Y 680.524,Z 396.45,A -85,B 0,C 180,E1 31466.363,E2 31466.363} C_VEL
LIN {X 0,Y 680.488,Z 396.464,A -85,B 0,C 180,E1 31463.337,E2 31463.337} C_VEL
LIN {X 0,Y 680.524,Z 396.455,A -85,B 0,C 180,E1 31460.381,E2 31460.381} C_VEL
LIN {X 0,Y 680.5,Z 396.461,A -85,B 0,C 180,E1 31457.27,E2 31457.27} C_VEL
LIN {X 0,Y 680.496,Z 396.503,A -85,B 0,C 180,E1 31457.077,E2 31457.077} C_VEL
LIN {X 0,Y 681.089,Z 398.661,A -85,B 0,C 180,E1 31456.891,E2 31456.891} C_VEL
LIN {X 0,Y 683.247,Z 401.566,A -85,B 0,C 180,E1 31456.654,E2 31456.654} C_VEL
LIN {X 0,Y 690.96,Z 412.714,A -85,B 0,C 180,E1 31455.816,E2 31455.816} C_VEL
LIN {X 0,Y 700.726,Z 427.339,A -85,B 0,C 180,E1 31454.792,E2 31454.792} C_VEL
LIN {X 0,Y 698.44,Z 631.493,A -85,B 0,C 180,E1 31452.138,E2 31452.138} C_VEL
LIN {X 0,Y 696.107,Z 856.745,A -85,B 0,C 180,E1 31449.303,E2 31449.303} C_VEL
LIN {X 0,Y 695.54,Z 887.245,A -85,B 0,C 180,E1 31448.862,E2 31448.862} C_VEL
LIN {X 0,Y 694.783,Z 912.229,A -85,B 0,C 180,E1 31448.352,E2 31448.352} C_VEL
LIN {X 0,Y 693.895,Z 937.894,A -85,B 0,C 180,E1 31447.678,E2 31447.678} C_VEL
LIN {X 0,Y 692.766,Z 964.789,A -85,B 0,C 180,E1 31446.79,E2 31446.79} C_VEL
LIN {X 0,Y 691.756,Z 986.072,A -85,B 0,C 180,E1 31445.958,E2 31445.958} C_VEL
LIN {X 0,Y 690.739,Z 1005.955,A -85,B 0,C 180,E1 31445.07,E2 31445.07} C_VEL
LIN {X 0,Y 689.668,Z 1025.744,A -85,B 0,C 180,E1 31444.073,E2 31444.073} C_VEL
LIN {X 0,Y 688.514,Z 1046.626,A -85,B 0,C 180,E1 31442.891,E2 31442.891} C_VEL
LIN {X 0,Y 687.057,Z 1071.374,A -85,B 0,C 180,E1 31441.296,E2 31441.296} C_VEL
LIN {X 0,Y 685.976,Z 1090.559,A -85,B 0,C 180,E1 31439.895,E2 31439.895} C_VEL
LIN {X 0,Y 684.948,Z 1109.472,A -85,B 0,C 180,E1 31438.364,E2 31438.364} C_VEL
LIN {X 0,Y 683.772,Z 1130.661,A -85,B 0,C 180,E1 31436.435,E2 31436.435} C_VEL
LIN {X 0,Y 682.96,Z 1147.179,A -85,B 0,C 180,E1 31434.748,E2 31434.748} C_VEL
LIN {X 0,Y 682.134,Z 1164.686,A -85,B 0,C 180,E1 31432.761,E2 31432.761} C_VEL
LIN {X 0,Y 681.457,Z 1180.528,A -85,B 0,C 180,E1 31430.703,E2 31430.703} C_VEL
LIN {X 0,Y 681.03,Z 1192.75,A -85,B 0,C 180,E1 31428.928,E2 31428.928} C_VEL
LIN {X 0,Y 680.635,Z 1205.144,A -85,B 0,C 180,E1 31426.905,E2 31426.905} C_VEL
LIN {X 0,Y 680.338,Z 1217.059,A -85,B 0,C 180,E1 31424.638,E2 31424.638} C_VEL
LIN {X 0,Y 680.162,Z 1225.626,A -85,B 0,C 180,E1 31422.734,E2 31422.734} C_VEL
LIN {X 0,Y 680.027,Z 1232.599,A -85,B 0,C 180,E1 31420.929,E2 31420.929} C_VEL
LIN {X 0,Y 679.931,Z 1238.186,A -85,B 0,C 180,E1 31419.219,E2 31419.219} C_VEL
LIN {X 0,Y 679.923,Z 1243.275,A -85,B 0,C 180,E1 31417.346,E2 31417.346} C_VEL
LIN {X 0,Y 679.918,Z 1247.858,A -85,B 0,C 180,E1 31415.058,E2 31415.058} C_VEL
LIN {X 0,Y 679.913,Z 1250.576,A -85,B 0,C 180,E1 31412.862,E2 31412.862} C_VEL
LIN {X 0,Y 679.878,Z 1251.726,A -85,B 0,C 180,E1 31411.007,E2 31411.007} C_VEL
LIN {X 0,Y 679.864,Z 1251.838,A -85,B 0,C 180,E1 31409.322,E2 31409.322} C_VEL
LIN {X 0,Y 679.903,Z 1250.979,A -85,B 0,C 180,E1 31407.552,E2 31407.552} C_VEL
LIN {X 0,Y 679.913,Z 1248.861,A -85,B 0,C 180,E1 31405.526,E2 31405.526} C_VEL
LIN {X 0,Y 679.926,Z 1244.819,A -85,B 0,C 180,E1 31403.24,E2 31403.24} C_VEL
LIN {X 0,Y 679.939,Z 1239.201,A -85,B 0,C 180,E1 31401.029,E2 31401.029} C_VEL
LIN {X 0,Y 680.015,Z 1233.199,A -85,B 0,C 180,E1 31399.148,E2 31399.148} C_VEL
LIN {X 0,Y 680.145,Z 1226.324,A -85,B 0,C 180,E1 31397.344,E2 31397.344} C_VEL
LIN {X 0,Y 680.308,Z 1218.267,A -85,B 0,C 180,E1 31395.528,E2 31395.528} C_VEL
LIN {X 0,Y 680.537,Z 1208.032,A -85,B 0,C 180,E1 31393.524,E2 31393.524} C_VEL
LIN {X 0,Y 680.997,Z 1193.866,A -85,B 0,C 180,E1 31391.151,E2 31391.151} C_VEL
LIN {X 0,Y 681.433,Z 1181.114,A -85,B 0,C 180,E1 31389.288,E2 31389.288} C_VEL
LIN {X 0,Y 682.033,Z 1166.749,A -85,B 0,C 180,E1 31387.409,E2 31387.409} C_VEL
LIN {X 0,Y 682.886,Z 1148.776,A -85,B 0,C 180,E1 31385.333,E2 31385.333} C_VEL
LIN {X 0,Y 683.694,Z 1132.252,A -85,B 0,C 180,E1 31383.632,E2 31383.632} C_VEL
LIN {X 0,Y 684.776,Z 1112.855,A -85,B 0,C 180,E1 31381.83,E2 31381.83} C_VEL
LIN {X 0,Y 685.875,Z 1092.434,A -85,B 0,C 180,E1 31380.16,E2 31380.16} C_VEL
LIN {X 0,Y 686.938,Z 1073.823,A -85,B 0,C 180,E1 31378.787,E2 31378.787} C_VEL
LIN {X 0,Y 688.201,Z 1051.824,A -85,B 0,C 180,E1 31377.331,E2 31377.331} C_VEL
LIN {X 0,Y 689.543,Z 1028.072,A -85,B 0,C 180,E1 31375.961,E2 31375.961} C_VEL
LIN {X 0,Y 690.656,Z 1007.537,A -85,B 0,C 180,E1 31374.915,E2 31374.915} C_VEL
LIN {X 0,Y 691.633,Z 988.526,A -85,B 0,C 180,E1 31374.056,E2 31374.056} C_VEL
LIN {X 0,Y 692.593,Z 968.28,A -85,B 0,C 180,E1 31373.25,E2 31373.25} C_VEL
LIN {X 0,Y 693.561,Z 945.3,A -85,B 0,C 180,E1 31372.46,E2 31372.46} C_VEL
LIN {X 0,Y 694.597,Z 918.719,A -85,B 0,C 180,E1 31371.712,E2 31371.712} C_VEL
LIN {X 0,Y 695.368,Z 892.814,A -85,B 0,C 180,E1 31371.15,E2 31371.15} C_VEL
LIN {X 0,Y 695.946,Z 867.809,A -85,B 0,C 180,E1 31370.749,E2 31370.749} C_VEL
LIN {X 0,Y 698.327,Z 641.745,A -85,B 0,C 180,E1 31367.902,E2 31367.902} C_VEL
LIN {X 0,Y 700.647,Z 434.74,A -85,B 0,C 180,E1 31365.217,E2 31365.217} C_VEL
LIN {X 0,Y 700.548,Z 426.842,A -85,B 0,C 180,E1 31365.097,E2 31365.097} C_VEL
LIN {X 0,Y 686.611,Z 406.259,A -85,B 0,C 180,E1 31363.623,E2 31363.623} C_VEL
LIN {X 0,Y 682.929,Z 401.266,A -85,B 0,C 180,E1 31363.223,E2 31363.223} C_VEL
LIN {X 0,Y 680.959,Z 398.304,A -85,B 0,C 180,E1 31363.002,E2 31363.002} C_VEL
LIN {X 0,Y 680.504,Z 396.461,A -85,B 0,C 180,E1 31362.818,E2 31362.818} C_VEL
LIN {X 0,Y 680.505,Z 396.466,A -85,B 0,C 180,E1 31359.839,E2 31359.839} C_VEL
LIN {X 0,Y 680.51,Z 396.466,A -85,B 0,C 180,E1 31356.934,E2 31356.934} C_VEL
LIN {X 0,Y 680.51,Z 396.447,A -85,B 0,C 180,E1 31353.882,E2 31353.882} C_VEL
LIN {X 0,Y 680.515,Z 396.446,A -85,B 0,C 180,E1 31350.85,E2 31350.85} C_VEL
LIN {X 0,Y 680.516,Z 396.458,A -85,B 0,C 180,E1 31347.76,E2 31347.76} C_VEL
LIN {X 0,Y 680.518,Z 396.449,A -85,B 0,C 180,E1 31344.663,E2 31344.663} C_VEL
LIN {X 0,Y 680.514,Z 396.452,A -85,B 0,C 180,E1 31341.551,E2 31341.551} C_VEL
LIN {X 0,Y 680.523,Z 396.459,A -85,B 0,C 180,E1 31338.504,E2 31338.504} C_VEL
LIN {X 0,Y 680.517,Z 396.443,A -85,B 0,C 180,E1 31335.423,E2 31335.423} C_VEL
LIN {X 0,Y 680.523,Z 396.463,A -85,B 0,C 180,E1 31332.288,E2 31332.288} C_VEL
LIN {X 0,Y 680.507,Z 396.438,A -85,B 0,C 180,E1 31329.106,E2 31329.106} C_VEL
LIN {X 0,Y 680.523,Z 396.465,A -85,B 0,C 180,E1 31326.073,E2 31326.073} C_VEL
LIN {X 0,Y 680.509,Z 396.435,A -85,B 0,C 180,E1 31322.948,E2 31322.948} C_VEL
LIN {X 0,Y 680.529,Z 396.465,A -85,B 0,C 180,E1 31319.832,E2 31319.832} C_VEL
LIN {X 0,Y 680.508,Z 396.433,A -85,B 0,C 180,E1 31316.715,E2 31316.715} C_VEL
LIN {X 0,Y 680.518,Z 396.465,A -85,B 0,C 180,E1 31313.673,E2 31313.673} C_VEL
LIN {X 0,Y 680.51,Z 396.437,A -85,B 0,C 180,E1 31310.528,E2 31310.528} C_VEL
LIN {X 0,Y 680.509,Z 396.466,A -85,B 0,C 180,E1 31307.526,E2 31307.526} C_VEL
LIN {X 0,Y 680.509,Z 396.446,A -85,B 0,C 180,E1 31304.314,E2 31304.314} C_VEL
LIN {X 0,Y 680.507,Z 396.461,A -85,B 0,C 180,E1 31301.318,E2 31301.318} C_VEL
LIN {X 0,Y 680.508,Z 396.456,A -85,B 0,C 180,E1 31298.086,E2 31298.086} C_VEL
LIN {X 0,Y 680.505,Z 396.448,A -85,B 0,C 180,E1 31295.058,E2 31295.058} C_VEL
